# B&R Automation Studio project TD52 (part 64)

```c
    /* Switch: '<S85>/Switch' incorporates:
     *  RelationalOperator: '<S85>/UpperRelop'
     */
    if (rtb_deltafalllimit_h0 < rtb_Saturation_e) {
      rtb_Sum1_dh = rtb_Saturation_e;
    } else {
      rtb_Sum1_dh = rtb_deltafalllimit_h0;
    }

    /* End of Switch: '<S85>/Switch' */
  }

  /* End of Switch: '<S85>/Switch2' */

  /* Sum: '<S81>/Difference Inputs2' incorporates:
   *  Delay: '<S81>/Delay'
   */
  rtb_Saturation_e = rtb_Sum1_dh + Gen2_ref_DWork->Delay_DSTATE_h;

  /* Switch: '<S77>/Switch' */
  if (rtb_LogicalOperator2_p1) {
    /* Switch: '<S77>/Switch2' */
    if (Gen2_ref_B->BusInput3.traj.bRateLimRejStepSizeDep) {
      rtb_Sum1_dh = rtb_Gain_i;
    } else {
      rtb_Sum1_dh = rtb_Saturation_e;
    }

    /* End of Switch: '<S77>/Switch2' */
  } else {
    rtb_Sum1_dh = rtb_p1HP;
  }

  /* End of Switch: '<S77>/Switch' */

  /* MinMax: '<S77>/MinMax1' */
  if ((rtb_p1HP >= rtb_Sum1_dh) || rtIsNaN(rtb_Sum1_dh)) {
    rtb_MinMax1_g = rtb_p1HP;
  } else {
    rtb_MinMax1_g = rtb_Sum1_dh;
  }

  /* End of MinMax: '<S77>/MinMax1' */

  /* Abs: '<S23>/Abs1' */
  rtb_Sum1_dh = fabs(Gen2_ref_B->BusInput3.traj.rPrTriggerLargeRej);

  /* Switch: '<S23>/Switch1' incorporates:
   *  RelationalOperator: '<S23>/Relational Operator3'
   *  Sum: '<S23>/Sum7'
   */
  if (rtb_Gain_kl - rtb_p1HP > rtb_Sum1_dh) {
    rtb_Switch1_lk = Gen2_ref_B->BusInput3.traj.rTi_BDC_rej_CBV;
  } else {
    rtb_Switch1_lk = Gen2_ref_B->BusInput3.traj.rTi_BDC;
  }

  /* End of Switch: '<S23>/Switch1' */

  /* Product: '<S23>/Product1' */
  rtb_Product1_bc = Gen2_ref_B->BusInput3.traj.rFactTi_BDC_CBV * rtb_Switch1_lk;

  /* Switch: '<S1>/Switch13' incorporates:
   *  DataTypeConversion: '<S4>/Data Type Conversion16'
   */
  if (Gen2_ref_B->BusInput3.bdcMisc.bUseNsetBDC) {
    rtb_Switch13 = Gen2_ref_B->BusInput.rN_Set;
  } else {
    rtb_Switch13 = Gen2_ref_B->BusInput3.eng.rN_Nom;
  }

  /* End of Switch: '<S1>/Switch13' */

  /* Sum: '<S23>/Sum4' incorporates:
   *  Sum: '<S133>/Sum'
   */
  rtb_Switch1_kk = rtb_DataTypeConversion15 - rtb_Switch13;

  /* MATLAB Function: '<S23>/ref traj' incorporates:
   *  MATLAB Function: '<S431>/ref traj'
   *  Sum: '<S23>/Sum4'
   */
  if ((!Gen2_ref_DWork->x_not_empty_n) || rtb_LogicalOperator2_dc) {
    Gen2_ref_DWork->x_e = rtb_Gain_kl;
    Gen2_ref_DWork->x_not_empty_n = true;
    Gen2_ref_DWork->x0 = rtb_Gain_kl;
    Gen2_ref_DWork->x1 = rtb_Gain_kl;
    Gen2_ref_DWork->x2 = rtb_Gain_kl;
    Gen2_ref_DWork->x3 = rtb_Gain_kl;
    Gen2_ref_DWork->x4 = rtb_Gain_kl;
  }

  if (Gen2_ref_B->BusInput3.eng.Ts >= 0.01) {
    Ts_tmp = Gen2_ref_B->BusInput3.eng.Ts;
  } else {
    Ts_tmp = 0.01;
  }

  delta_y = rtb_MinMax1_h - rtb_Gain_kl;
  if (delta_y > Gen2_ref_B->BusInput3.traj.rThrshSwTbdcUp) {
    rtb_Switch2_j0 = Gen2_ref_B->BusInput3.traj.rTi_BDC_up;
  } else {
    rtb_Switch2_j0 = Gen2_ref_B->BusInput3.traj.rTi_BDC;
  }

  if (Gen2_ref_B->BusInput3.traj.bLimitFFcmdTV) {
    if ((rtb_Sum11 >= rtb_MinMax1_h) || rtIsNaN(rtb_MinMax1_h)) {
      FILT_IN = rtb_Sum11;
    } else {
      FILT_IN = rtb_MinMax1_h;
    }
  } else {
    FILT_IN = rtb_Sum11;
  }

  rtb_LogicalOperator5_g_tmp = rtIsNaN(Ts_tmp);
  if ((rtb_Switch2_j0 >= Ts_tmp) || rtb_LogicalOperator5_g_tmp) {
    r = rtb_Switch2_j0;
  } else {
    r = Ts_tmp;
  }

  rtb_Switch2_a = FILT_IN - Gen2_ref_DWork->x0;
  u0 = 1.0 / r * rtb_Switch2_a;
  if ((Gen2_ref_B->BusInput3.traj.rTi_BDC >= Ts_tmp) ||
      rtb_LogicalOperator5_g_tmp) {
    FILT_IN = Gen2_ref_B->BusInput3.traj.rTi_BDC;
  } else {
    FILT_IN = Ts_tmp;
  }

  u1 = 1.0 / FILT_IN * rtb_Switch2_a;
  if ((u0 >= u1) || rtIsNaN(u1)) {
    u1 = u0;
  }

  rtb_Sum10 = u1 * Ts_tmp + Gen2_ref_DWork->x0;
  if (Gen2_ref_B->BusInput3.traj.bLimitFFcmdCBV) {
    if ((rtb_Sum7_l5 >= rtb_MinMax1_g) || rtIsNaN(rtb_MinMax1_g)) {
      FILT_IN = rtb_Sum7_l5;
    } else {
      FILT_IN = rtb_MinMax1_g;
    }
  } else {
    FILT_IN = rtb_Sum7_l5;
  }

  if (rtb_Switch1_kk > 0.0) {
    if ((rtb_Switch2_j0 >= Ts_tmp) || rtb_LogicalOperator5_g_tmp) {
      r = rtb_Switch2_j0;
    } else {
      r = Ts_tmp;
    }

    rtb_Switch2_a = FILT_IN - Gen2_ref_DWork->x1;
    u0 = 1.0 / r * rtb_Switch2_a;
    if ((rtb_Product1_bc >= Ts_tmp) || rtb_LogicalOperator5_g_tmp) {
      FILT_IN = rtb_Product1_bc;
    } else {
      FILT_IN = Ts_tmp;
    }

    FILT_IN = 1.0 / FILT_IN * rtb_Switch2_a;
    if ((u0 >= FILT_IN) || rtIsNaN(FILT_IN)) {
      FILT_IN = u0;
    }
  } else {
    if ((rtb_Switch2_j0 >= Ts_tmp) || rtb_LogicalOperator5_g_tmp) {
      r = rtb_Switch2_j0;
    } else {
      r = Ts_tmp;
    }

    rtb_Switch2_a = FILT_IN - Gen2_ref_DWork->x1;
    u0 = 1.0 / r * rtb_Switch2_a;
    if ((Gen2_ref_B->BusInput3.traj.rTi_BDC >= Ts_tmp) ||
        rtb_LogicalOperator5_g_tmp) {
      FILT_IN = Gen2_ref_B->BusInput3.traj.rTi_BDC;
    } else {
      FILT_IN = Ts_tmp;
    }

    FILT_IN = 1.0 / FILT_IN * rtb_Switch2_a;
    if ((u0 >= FILT_IN) || rtIsNaN(FILT_IN)) {
      FILT_IN = u0;
    }
  }

  rtb_Switch2_h1 = FILT_IN * Ts_tmp + Gen2_ref_DWork->x1;
  if ((rtb_Switch2_j0 >= Ts_tmp) || rtb_LogicalOperator5_g_tmp) {
    r = rtb_Switch2_j0;
  } else {
    r = Ts_tmp;
  }

  rtb_Switch2_a = rtb_MinMax1_h - Gen2_ref_DWork->x2;
  u0 = 1.0 / r * rtb_Switch2_a;
  if ((Gen2_ref_B->BusInput3.traj.rTi_BDC >= Ts_tmp) ||
      rtb_LogicalOperator5_g_tmp) {
    FILT_IN = Gen2_ref_B->BusInput3.traj.rTi_BDC;
  } else {
    FILT_IN = Ts_tmp;
  }

  u1 = 1.0 / FILT_IN * rtb_Switch2_a;
  if ((u0 >= u1) || rtIsNaN(u1)) {
    u1 = u0;
  }

  rtb_Switch2_lu = u1 * Ts_tmp + Gen2_ref_DWork->x2;
  if ((rtb_Switch2_j0 >= Ts_tmp) || rtb_LogicalOperator5_g_tmp) {
    r = rtb_Switch2_j0;
  } else {
    r = Ts_tmp;
  }

  rtb_Switch2_a = rtb_MinMax1_g - Gen2_ref_DWork->x3;
  u0 = 1.0 / r * rtb_Switch2_a;
  rtb_bCBV_min = !rtb_LogicalOperator5_g_tmp;
  if ((!(rtb_Product1_bc >= Ts_tmp)) && rtb_bCBV_min) {
    rtb_Product1_bc = Ts_tmp;
  }

  u1 = 1.0 / rtb_Product1_bc * rtb_Switch2_a;
  if ((u0 >= u1) || rtIsNaN(u1)) {
    u1 = u0;
  }

  rtb_Divide3_k = u1 * Ts_tmp + Gen2_ref_DWork->x3;
  if ((rtb_Switch2_j0 >= Ts_tmp) || rtb_LogicalOperator5_g_tmp) {
    r = rtb_Switch2_j0;
  } else {
    r = Ts_tmp;
  }

  rtb_Switch2_a = rtb_Sum11 - Gen2_ref_DWork->x_e;
  u0 = 1.0 / r * rtb_Switch2_a;
  if ((Gen2_ref_B->BusInput3.traj.rTi_BDC >= Ts_tmp) ||
      rtb_LogicalOperator5_g_tmp) {
    FILT_IN = Gen2_ref_B->BusInput3.traj.rTi_BDC;
  } else {
    FILT_IN = Ts_tmp;
  }

  FILT_IN = 1.0 / FILT_IN * rtb_Switch2_a;
  if ((u0 >= FILT_IN) || rtIsNaN(FILT_IN)) {
    FILT_IN = u0;
  }

  if (FILT_IN > 0.0) {
    u0 = FILT_IN * Ts_tmp + Gen2_ref_DWork->x_e;
    rtb_Product1_bc = rtb_Gain_kl + Gen2_ref_B->BusInput3.traj.rPrR_delta_p2s;
    if ((u0 <= rtb_Product1_bc) || rtIsNaN(rtb_Product1_bc)) {
      rtb_Product1_bc = u0;
    }
  } else {
    u0 = FILT_IN * Ts_tmp + Gen2_ref_DWork->x_e;
    rtb_Product1_bc = rtb_Gain_kl - Gen2_ref_B->BusInput3.traj.rPrR_delta_p2s;
    if ((u0 >= rtb_Product1_bc) || rtIsNaN(rtb_Product1_bc)) {
      rtb_Product1_bc = u0;
    }
  }

  if ((!(rtb_Switch2_j0 >= Ts_tmp)) && rtb_bCBV_min) {
    rtb_Switch2_j0 = Ts_tmp;
  }

  rtb_Switch2_a = rtb_Sum7_l5 - Gen2_ref_DWork->x4;
  u0 = 1.0 / rtb_Switch2_j0 * rtb_Switch2_a;
  if ((!(rtb_Switch1_lk >= Ts_tmp)) && rtb_bCBV_min) {
    rtb_Switch1_lk = Ts_tmp;
  }

  u1 = 1.0 / rtb_Switch1_lk * rtb_Switch2_a;
  if (FILT_IN > 0.0) {
    if ((u0 >= u1) || rtIsNaN(u1)) {
      u1 = u0;
    }

    u0 = u1 * Ts_tmp + Gen2_ref_DWork->x4;
    rtb_Switch2_j0 = rtb_Gain_kl + Gen2_ref_B->BusInput3.traj.rPrR_delta_p2s;
    if ((u0 <= rtb_Switch2_j0) || rtIsNaN(rtb_Switch2_j0)) {
      rtb_Switch2_j0 = u0;
    }
  } else {
    if ((u0 >= u1) || rtIsNaN(u1)) {
      u1 = u0;
    }

    rtb_Switch2_j0 = u1 * Ts_tmp + Gen2_ref_DWork->x4;
  }

  Gen2_ref_DWork->x_e = rtb_Product1_bc;
  Gen2_ref_DWork->x0 = rtb_Sum10;
  Gen2_ref_DWork->x1 = rtb_Switch2_h1;
  Gen2_ref_DWork->x2 = rtb_Switch2_lu;
  Gen2_ref_DWork->x3 = rtb_Divide3_k;
  Gen2_ref_DWork->x4 = rtb_Switch2_j0;

  /* Product: '<S64>/delta rise limit' incorporates:
   *  Constant: '<S23>/Constant4'
   *  SampleTimeMath: '<S64>/sample time'
   *
   * About '<S64>/sample time':
   *  y = K where K = ( w * Ts )
   */
  rtb_Sum1_dh = 100000.0;

  /* S-Function (sfix_look1_dyn): '<S23>/Lookup Table Dynamic1' */
  /* Dynamic Look-Up Table Block: '<S23>/Lookup Table Dynamic1'
   * Input0  Data Type:  Floating Point real_T
   * Input1  Data Type:  Floating Point real_T
   * Input2  Data Type:  Floating Point real_T
   * Output0 Data Type:  Floating Point real_T
   * Lookup Method: Linear_Endpoint
   *
   */
  LookUp_real_T_real_T( &(rtb_MinMax_a),
                       &Gen2_ref_B->BusInput3.traj.rRateLimTVdpctrl[0],
                       rtb_Gain_kl, &rtb_Gain1_eu[0], 4U, inst);

  /* Abs: '<S23>/Abs3' */
  rtb_Switch1_lk = fabs(rtb_MinMax_a);

  /* Product: '<S63>/delta rise limit' incorporates:
   *  SampleTimeMath: '<S63>/sample time'
   *
   * About '<S63>/sample time':
   *  y = K where K = ( w * Ts )
   */
  rtb_MinMax_a = rtb_Switch1_lk * 0.01;

  /* Switch: '<S23>/Switch2' incorporates:
   *  Delay: '<S23>/Delay'
   *  Switch: '<S23>/Switch4'
   */
  if (Gen2_ref_DWork->Delay_DSTATE_lv) {
    FILT_IN = rtb_Product2;
  } else if (Gen2_ref_B->BusInput3.traj.bFactInitResetTVdp) {
    /* Sum: '<S23>/Sum' incorporates:
     *  MATLAB Function: '<S23>/ref traj'
     *  Switch: '<S23>/Switch4'
     */
    FILT_IN = Gen2_ref_B->BusInput3.traj.rPrR_TC_LP_min - rtb_Divide3_k;

    /* Saturate: '<S23>/Saturation' incorporates:
     *  Switch: '<S23>/Switch4'
     */
    if (FILT_IN > 1.0) {
      FILT_IN = 1.0;
    } else if (FILT_IN < 0.0) {
      FILT_IN = 0.0;
    }

    /* End of Saturate: '<S23>/Saturation' */
  } else {
    /* Switch: '<S23>/Switch4' incorporates:
     *  Constant: '<S23>/Constant2'
     */
    FILT_IN = 0.0;
  }

  /* End of Switch: '<S23>/Switch2' */

  /* Logic: '<S23>/Logical Operator4' incorporates:
   *  Constant: '<S23>/Constant1'
   *  MATLAB Function: '<S23>/ref traj'
   *  RelationalOperator: '<S23>/Relational Operator2'
   *  Sum: '<S23>/Sum4'
   */
  rtb_LogicalOperator2_p1 = (((rtb_Sum11 - rtb_Gain_kl >
    Gen2_ref_B->BusInput3.traj.rPr_delta_p2s_resetTVdp) || (delta_y >
    Gen2_ref_B->BusInput3.traj.rPr_delta_p2s_resetTVdp) ||
    rtb_LogicalOperator2_dc) && (rtb_Switch1_kk <= 0.0));

  /* Abs: '<S23>/Abs' incorporates:
   *  Sum: '<S23>/Sum4'
   */
  rtb_Switch2_a = fabs(rtb_Switch1_kk);

  /* Outputs for Atomic SubSystem: '<S23>/TON_1' */
  /* Logic: '<S23>/Logical Operator5' incorporates:
   *  Logic: '<S23>/Logical Operator6'
   *  RelationalOperator: '<S23>/Relational Operator'
   */
  Gen2_ref_TON_1(((!rtb_LogicalOperator2_p1) && (rtb_Switch2_a <=
    Gen2_ref_B->BusInput3.traj.rN_ssTVdpCtrl)),
                 Gen2_ref_B->BusInput3.traj.rT_TON_TVdpCtrl, &Gen2_ref_B->TON_1,
                 &Gen2_ref_DWork->TON_1, inst);

  /* End of Outputs for SubSystem: '<S23>/TON_1' */

  /* Switch: '<S53>/Switch' incorporates:
   *  Switch: '<S53>/Switch1'
   *  UnitDelay: '<S53>/Unit Delay4'
   */
  if (!rtb_LogicalOperator2_p1) {
    rtb_LogicalOperator2_p1 = ((!Gen2_ref_B->TON_1.LogicalOperator3) &&
      Gen2_ref_DWork->UnitDelay4_DSTATE_o);
  }

  /* End of Switch: '<S53>/Switch' */

  /* Logic: '<S23>/Logical Operator1' */
  rtb_LogicalOperator1_a0 = (rtb_LogicalOperator || rtb_LogicalOperator2_p1);

  /* Delay: '<S63>/Delay' */
  Gen2_ref_DWork->icLoad_g = ((((Gen2_ref_PrevZCSigState->Delay_Reset_ZCE_k2 ==
    1) != (int32_T)rtb_LogicalOperator1_a0) &&
    (Gen2_ref_PrevZCSigState->Delay_Reset_ZCE_k2 != 3)) ||
    rtb_LogicalOperator1_a0 || Gen2_ref_DWork->icLoad_g);
  Gen2_ref_PrevZCSigState->Delay_Reset_ZCE_k2 = rtb_LogicalOperator1_a0;
  if (Gen2_ref_DWork->icLoad_g) {
    Gen2_ref_DWork->Delay_DSTATE_c = FILT_IN;
  }

  /* Switch: '<S63>/etaVolConst' */
  if (!rtb_LogicalOperator1_a0) {
    FILT_IN = rtb_Product2;
  }

  /* End of Switch: '<S63>/etaVolConst' */

  /* Sum: '<S63>/Difference Inputs1' incorporates:
   *  Delay: '<S63>/Delay'
   */
  rtb_deltafalllimit_h0 = FILT_IN - Gen2_ref_DWork->Delay_DSTATE_c;

  /* Switch: '<S102>/Switch2' incorporates:
   *  RelationalOperator: '<S102>/LowerRelop1'
   */
  if (!(rtb_deltafalllimit_h0 > rtb_MinMax_a)) {
    /* Product: '<S63>/delta fall limit' incorporates:
     *  Gain: '<S23>/Gain4'
     *  SampleTimeMath: '<S63>/sample time'
     *
     * About '<S63>/sample time':
     *  y = K where K = ( w * Ts )
     */
    rtb_Switch1_lk = -rtb_Switch1_lk * 0.01;

    /* Switch: '<S102>/Switch' incorporates:
     *  RelationalOperator: '<S102>/UpperRelop'
     */
    if (rtb_deltafalllimit_h0 < rtb_Switch1_lk) {
      rtb_MinMax_a = rtb_Switch1_lk;
    } else {
      rtb_MinMax_a = rtb_deltafalllimit_h0;
    }

    /* End of Switch: '<S102>/Switch' */
  }

  /* End of Switch: '<S102>/Switch2' */

  /* Sum: '<S63>/Difference Inputs2' incorporates:
   *  Delay: '<S63>/Delay'
   */
  rtb_deltafalllimit_h0 = rtb_MinMax_a + Gen2_ref_DWork->Delay_DSTATE_c;

  /* Switch: '<S23>/Switch3' */
  if (rtb_LogicalOperator) {
    rtb_MinMax_a = rtb_Product2;
  } else {
    rtb_MinMax_a = rtb_deltafalllimit_h0;
  }

  /* End of Switch: '<S23>/Switch3' */

  /* Saturate: '<S23>/Saturation2' */
  if (rtb_MinMax_a <= 0.0) {
    rtb_Switch2_a = 0.0;
  } else {
    rtb_Switch2_a = rtb_MinMax_a;
  }

  /* End of Saturate: '<S23>/Saturation2' */

  /* Delay: '<S64>/Delay' incorporates:
   *  Constant: '<S23>/Constant3'
   */
  Gen2_ref_DWork->icLoad_c1 = ((((Gen2_ref_PrevZCSigState->Delay_Reset_ZCE_a ==
    1) != (int32_T)rtb_LogicalOperator2_dc) &&
    (Gen2_ref_PrevZCSigState->Delay_Reset_ZCE_a != 3)) ||
    rtb_LogicalOperator2_dc || Gen2_ref_DWork->icLoad_c1);
  Gen2_ref_PrevZCSigState->Delay_Reset_ZCE_a = rtb_LogicalOperator2_dc;
  if (Gen2_ref_DWork->icLoad_c1) {
    Gen2_ref_DWork->Delay_DSTATE_i = 0.0;
  }

  /* Switch: '<S64>/etaVolConst' incorporates:
   *  Constant: '<S23>/Constant3'
   */
  if (rtb_LogicalOperator2_dc) {
    FILT_IN = 0.0;
  } else {
    FILT_IN = rtb_Switch2_a;
  }

  /* End of Switch: '<S64>/etaVolConst' */

  /* Sum: '<S64>/Difference Inputs1' incorporates:
   *  Delay: '<S64>/Delay'
   */
  rtb_Switch1_lk = FILT_IN - Gen2_ref_DWork->Delay_DSTATE_i;

  /* Switch: '<S103>/Switch2' incorporates:
   *  RelationalOperator: '<S103>/LowerRelop1'
   */
  if (!(rtb_Switch1_lk > 100000.0)) {
    /* Product: '<S64>/delta fall limit' incorporates:
     *  Abs: '<S23>/Abs2'
     *  Gain: '<S23>/Gain7'
     *  SampleTimeMath: '<S64>/sample time'
     *
     * About '<S64>/sample time':
     *  y = K where K = ( w * Ts )
     */
    FILT_IN = -fabs(Gen2_ref_B->BusInput3.traj.rRateResetTVdpctrl) * 0.01;

    /* Switch: '<S103>/Switch' incorporates:
     *  RelationalOperator: '<S103>/UpperRelop'
     */
    if (rtb_Switch1_lk < FILT_IN) {
      rtb_Sum1_dh = FILT_IN;
    } else {
      rtb_Sum1_dh = rtb_Switch1_lk;
    }

    /* End of Switch: '<S103>/Switch' */
  }

  /* End of Switch: '<S103>/Switch2' */

  /* Sum: '<S64>/Difference Inputs2' incorporates:
   *  Delay: '<S64>/Delay'
   */
  rtb_Switch1_lk = rtb_Sum1_dh + Gen2_ref_DWork->Delay_DSTATE_i;

  /* Sum: '<S23>/Sum5' incorporates:
   *  MATLAB Function: '<S23>/ref traj'
   */
  FILT_IN = rtb_Switch2_h1 + rtb_Switch1_lk;

  /* Switch: '<S54>/Switch2' incorporates:
   *  RelationalOperator: '<S54>/LowerRelop1'
   *  RelationalOperator: '<S54>/UpperRelop'
   *  Switch: '<S54>/Switch'
   */
  if (FILT_IN > rtb_Switch2_oou) {
    rtb_Switch2_h1 = rtb_Switch2_oou;
  } else if (FILT_IN < Gen2_ref_B->BusInput3.traj.rPrMinRefp2ff) {
    /* Switch: '<S54>/Switch' */
    rtb_Switch2_h1 = Gen2_ref_B->BusInput3.traj.rPrMinRefp2ff;
  } else {
    rtb_Switch2_h1 = FILT_IN;
  }

  /* End of Switch: '<S54>/Switch2' */

  /* Switch: '<S60>/Switch2' incorporates:
   *  MATLAB Function: '<S23>/ref traj'
   *  RelationalOperator: '<S60>/LowerRelop1'
   *  RelationalOperator: '<S60>/UpperRelop'
   *  Switch: '<S60>/Switch'
   */
  if (rtb_Switch2_lu > Gen2_ref_B->BusInput3.traj.rPr_p2s_max) {
    rtb_Switch2_lu = Gen2_ref_B->BusInput3.traj.rPr_p2s_max;
  } else if (rtb_Switch2_lu < Gen2_ref_B->BusInput3.traj.rPr_p2s_min) {
    /* Switch: '<S60>/Switch' */
    rtb_Switch2_lu = Gen2_ref_B->BusInput3.traj.rPr_p2s_min;
  }

  /* End of Switch: '<S60>/Switch2' */

  /* Sum: '<S23>/Sum2' incorporates:
   *  MATLAB Function: '<S23>/ref traj'
   */
  FILT_IN = rtb_Divide3_k + rtb_Switch2_a;

  /* Switch: '<S59>/Switch2' incorporates:
   *  RelationalOperator: '<S59>/LowerRelop1'
   *  RelationalOperator: '<S59>/UpperRelop'
   *  Switch: '<S59>/Switch'
   */
  if (FILT_IN > Gen2_ref_B->BusInput3.traj.rPr_p2s_max) {
    rtb_Sum1_dh = Gen2_ref_B->BusInput3.traj.rPr_p2s_max;
  } else if (FILT_IN < Gen2_ref_B->BusInput3.traj.rPrMinRefp2ff) {
    /* Switch: '<S59>/Switch' */
    rtb_Sum1_dh = Gen2_ref_B->BusInput3.traj.rPrMinRefp2ff;
  } else {
    rtb_Sum1_dh = FILT_IN;
  }

  /* End of Switch: '<S59>/Switch2' */

  /* Abs: '<S68>/Abs' */
  rtb_Switch2_a = fabs(Gen2_ref_B->BusInput3.bdcMisc.rRefGainScheduleSL);

  /* Switch: '<S68>/Switch' incorporates:
   *  Constant: '<S68>/Constant2'
   *  RelationalOperator: '<S68>/Relational Operator'
   */
  if (2.2204460492503131E-16 >= rtb_Switch2_a) {
    FILT_IN = 2.2204460492503131E-16;
  } else {
    FILT_IN = Gen2_ref_B->BusInput3.bdcMisc.rRefGainScheduleSL;
  }

  /* End of Switch: '<S68>/Switch' */

  /* Abs: '<S67>/Abs' */
  rtb_Switch2_a = fabs(rtb_Switch13);

  /* Sum: '<S48>/Sum8' incorporates:
   *  Gain: '<S23>/Gain3'
   */
  rtb_Product4_d = 1.0E-5 * Gen2_ref_B->p2HP_filt.Switch - rtb_Switch2_oou;

  /* Switch: '<S67>/Switch' incorporates:
   *  Constant: '<S67>/Constant2'
   *  RelationalOperator: '<S67>/Relational Operator'
   */
  if (2.2204460492503131E-16 >= rtb_Switch2_a) {
    delta_y = 2.2204460492503131E-16;
  } else {
    delta_y = rtb_Switch13;
  }

  /* End of Switch: '<S67>/Switch' */

  /* Saturate: '<S48>/Saturation1' */
  if (rtb_Product4_d <= 0.0) {
    rtb_Product4_d = 0.0;
  }

  /* End of Saturate: '<S48>/Saturation1' */

  /* Product: '<S48>/Divide3' incorporates:
   *  DataTypeConversion: '<S48>/Data Type Conversion'
   *  Product: '<S48>/Divide2'
   *  RelationalOperator: '<S48>/Relational Operator2'
   */
  rtb_Divide3_k = (real_T)(Gen2_ref_B->BusInput3.LR.rN_LR_HardLim_norm > 1.0 /
    delta_y * rtb_DataTypeConversion15) * rtb_Product4_d;

  /* DiscreteIntegrator: '<S48>/Discrete-Time Integrator' */
  if (rtb_LogicalOperator2_dc ||
      (Gen2_ref_DWork->DiscreteTimeIntegrator_PrevRe_l != 0)) {
    Gen2_ref_DWork->DiscreteTimeIntegrator_DSTAT_ac = 0.0;
  }

  if (Gen2_ref_DWork->DiscreteTimeIntegrator_DSTAT_ac >= 1.0) {
    Gen2_ref_DWork->DiscreteTimeIntegrator_DSTAT_ac = 1.0;
  } else if (Gen2_ref_DWork->DiscreteTimeIntegrator_DSTAT_ac <= 0.0) {
    Gen2_ref_DWork->DiscreteTimeIntegrator_DSTAT_ac = 0.0;
  }

  /* Switch: '<S48>/Switch' incorporates:
   *  Constant: '<S48>/ON1'
   */
  if (Gen2_ref_B->BusInput3.SpeedCtrl.bSwitch_SurgeLine_LIMIT) {
    /* Sum: '<S48>/Sum12' incorporates:
     *  DiscreteIntegrator: '<S48>/Discrete-Time Integrator'
     *  Product: '<S48>/Product2'
     */
    rtb_Product4_d = rtb_Divide3_k *
      Gen2_ref_B->BusInput3.bdcMisc.rKpSurgeProtectSL +
      Gen2_ref_DWork->DiscreteTimeIntegrator_DSTAT_ac;

    /* Saturate: '<S48>/Saturation3' */
    if (rtb_Product4_d > 5.0) {
      rtb_Product4_d = 5.0;
    } else if (rtb_Product4_d < 0.0) {
      rtb_Product4_d = 0.0;
    }

    /* End of Saturate: '<S48>/Saturation3' */
  } else {
    rtb_Product4_d = 0.0;
  }

  /* End of Switch: '<S48>/Switch' */

  /* Product: '<S48>/Divide4' incorporates:
   *  Gain: '<S23>/Gain5'
   *  Product: '<S48>/Divide5'
   */
  rtb_Product4_d *= 1.0 / FILT_IN * (1.0E-5 * Gen2_ref_B->p2s_filt.Switch);

  /* Saturate: '<S23>/Saturation3' */
  if (rtb_MinMax_a >= 0.0) {
    rtb_Switch2_a = 0.0;
  } else {
    rtb_Switch2_a = rtb_MinMax_a;
  }

  /* End of Saturate: '<S23>/Saturation3' */

  /* Gain: '<S23>/Gain6' */
  rtb_Switch2_a = -rtb_Switch2_a;

  /* Sum: '<S23>/Sum9' incorporates:
   *  MATLAB Function: '<S23>/ref traj'
   *  Sum: '<S23>/Sum11'
   */
  rtb_Product1_bc = (rtb_Product1_bc + rtb_Switch2_a) + rtb_Product4_d;

  /* Switch: '<S56>/Switch2' incorporates:
   *  RelationalOperator: '<S56>/LowerRelop1'
   *  RelationalOperator: '<S56>/UpperRelop'
   *  Switch: '<S56>/Switch'
   */
  if (rtb_Product1_bc > Gen2_ref_B->BusInput3.traj.rPr_p2s_max) {
    /* BusCreator: '<S23>/Bus Creator1' */
    rtb_BusCreator1_ref_P2s_FB_TV = Gen2_ref_B->BusInput3.traj.rPr_p2s_max;
  } else if (rtb_Product1_bc < Gen2_ref_B->BusInput3.traj.rPr_p2s_min) {
    /* Switch: '<S56>/Switch' incorporates:
     *  BusCreator: '<S23>/Bus Creator1'
     */
    rtb_BusCreator1_ref_P2s_FB_TV = Gen2_ref_B->BusInput3.traj.rPr_p2s_min;
  } else {
    /* BusCreator: '<S23>/Bus Creator1' incorporates:
     *  Switch: '<S56>/Switch'
     */
    rtb_BusCreator1_ref_P2s_FB_TV = rtb_Product1_bc;
  }

  /* End of Switch: '<S56>/Switch2' */

  /* Sum: '<S23>/Sum1' incorporates:
   *  MATLAB Function: '<S23>/ref traj'
   */
  rtb_Product1_bc = rtb_Switch2_j0 + rtb_Switch1_lk;

  /* Switch: '<S55>/Switch2' incorporates:
   *  RelationalOperator: '<S55>/LowerRelop1'
   */
  if (!(rtb_Product1_bc > rtb_Switch2_oou)) {
    /* Switch: '<S55>/Switch' incorporates:
     *  RelationalOperator: '<S55>/UpperRelop'
     */
    if (rtb_Product1_bc < Gen2_ref_B->BusInput3.traj.rPrR_TC_LP_min) {
      rtb_Switch2_oou = Gen2_ref_B->BusInput3.traj.rPrR_TC_LP_min;
    } else {
      rtb_Switch2_oou = rtb_Product1_bc;
    }

    /* End of Switch: '<S55>/Switch' */
  }

  /* End of Switch: '<S55>/Switch2' */

  /* Sum: '<S23>/Sum10' incorporates:
   *  MATLAB Function: '<S23>/ref traj'
   *  Sum: '<S23>/Sum3'
   */
  rtb_Sum10 = (rtb_Sum10 + rtb_Switch2_a) + rtb_Product4_d;

  /* Switch: '<S57>/Switch2' incorporates:
   *  RelationalOperator: '<S57>/LowerRelop1'
   *  RelationalOperator: '<S57>/UpperRelop'
   *  Switch: '<S57>/Switch'
   */
  if (rtb_Sum10 > Gen2_ref_B->BusInput3.traj.rPr_p2s_max) {
    rtb_Switch2_jf = Gen2_ref_B->BusInput3.traj.rPr_p2s_max;
  } else if (rtb_Sum10 < Gen2_ref_B->BusInput3.traj.rPr_p2s_min) {
    /* Switch: '<S57>/Switch' */
    rtb_Switch2_jf = Gen2_ref_B->BusInput3.traj.rPr_p2s_min;
  } else {
    rtb_Switch2_jf = rtb_Sum10;
  }

  /* End of Switch: '<S57>/Switch2' */

  /* Outputs for Atomic SubSystem: '<S23>/Filter2' */
  /* UnitDelay: '<S23>/Unit Delay3' */
  Gen2_ref_Filter1(rtb_Switch2_jf, Gen2_ref_B->BusInput3.traj.rTiF_PrR_der,
                   Gen2_ref_DWork->UnitDelay3_DSTATE_gf, &Gen2_ref_B->Filter2,
                   &Gen2_ref_DWork->Filter2, inst);

  /* End of Outputs for SubSystem: '<S23>/Filter2' */

  /* Outputs for Atomic SubSystem: '<S23>/Filter1' */
  Gen2_ref_Filter1(rtb_Switch2_h1, Gen2_ref_B->BusInput3.traj.rTiF_PrR_der,
                   Gen2_ref_DWork->UnitDelay3_DSTATE_gf, &Gen2_ref_B->Filter1,
                   &Gen2_ref_DWork->Filter1, inst);

  /* End of Outputs for SubSystem: '<S23>/Filter1' */

  /* Outputs for Atomic SubSystem: '<S23>/Filter4' */
  Gen2_ref_Filter1(rtb_Switch2_lu, Gen2_ref_B->BusInput3.traj.rTiF_PrR_der,
                   Gen2_ref_DWork->UnitDelay3_DSTATE_gf, &Gen2_ref_B->Filter4,
                   &Gen2_ref_DWork->Filter4, inst);

  /* End of Outputs for SubSystem: '<S23>/Filter4' */

  /* BusCreator: '<S23>/Bus Creator1' */
  rtb_BusCreator1_ref_P2_FF = rtb_Sum1_dh;
  rtb_BusCreator1_ref_P2_FB_CBV = rtb_Switch2_oou;

  /* MultiPortSwitch: '<S24>/Multiport Switch' incorporates:
   *  BusCreator: '<S23>/Bus Creator1'
   */
  if ((int32_T)Gen2_ref_B->sf_MATLABFunction_f.y == 1) {
    rtb_Sum2_a1 = rtb_Switch2_jf;
  } else {
    rtb_Sum2_a1 = rtb_Switch2_lu;
  }

  /* End of MultiPortSwitch: '<S24>/Multiport Switch' */

  /* MATLAB Function: '<S44>/engine massflow2' incorporates:
   *  Gain: '<S1>/Gain9'
   *  Gain: '<S44>/rpm2rad1'
   */
  Gen2_ref_enginemassflow2(100000.0 * rtb_Sum2_a1, Gen2_ref_B->T2s_filt.Switch,
    0.10471975511965977 * rtb_Switch13, rtb_etaVolConst_lt,
    Gen2_ref_B->BusInput3.eng.rVol_Hub_Eng, &Gen2_ref_B->sf_enginemassflow2, inst);

  /* MultiPortSwitch: '<S24>/Multiport Switch1' incorporates:
   *  BusCreator: '<S23>/Bus Creator1'
   */
  if ((int32_T)Gen2_ref_B->sf_MATLABFunction_f.y == 1) {
    rtb_Sum2_a1 = Gen2_ref_B->Filter2.Switch1;
  } else {
    rtb_Sum2_a1 = Gen2_ref_B->Filter4.Switch1;
  }

  /* End of MultiPortSwitch: '<S24>/Multiport Switch1' */

  /* Gain: '<S1>/Gain10' */
  rtb_Switch2_oou = 100000.0 * rtb_Sum2_a1;

  /* DataTypeConversion: '<S155>/Data Type Conversion' */
  rtb_Sum2_a1 = Gen2_ref_B->BusInput3.bdcTv.bDynFFtv_ON;

  /* Product: '<S155>/Divide7' incorporates:
   *  Constant: '<S155>/R_air'
   */
  rtb_Product4_d = 287.15 * Gen2_ref_B->T2s_filt.Switch;

  /* Product: '<S155>/Divide6' */
  rtb_Product4_d = Gen2_ref_B->BusInput3.eng.rVol_im / rtb_Product4_d;

  /* Product: '<S155>/Divide8' */
  rtb_Switch2_oou = rtb_Switch2_oou * rtb_Sum2_a1 * rtb_Product4_d;

  /* Saturate: '<S44>/Saturation1' */
  if (Gen2_ref_B->BusInput3.eng.rNum_TV > 10.0) {
    rtb_Sum2_a1 = 10.0;
  } else if (Gen2_ref_B->BusInput3.eng.rNum_TV < 1.0) {
    rtb_Sum2_a1 = 1.0;
  } else {
    rtb_Sum2_a1 = Gen2_ref_B->BusInput3.eng.rNum_TV;
  }

  /* End of Saturate: '<S44>/Saturation1' */

  /* Product: '<S44>/Divide' incorporates:
   *  Sum: '<S44>/Sum3'
   */
  rtb_Divide_n0 = (Gen2_ref_B->sf_enginemassflow2.dm_e + rtb_Switch2_oou) /
    rtb_Sum2_a1;

  /* MultiPortSwitch: '<S24>/Multiport Switch2' incorporates:
   *  BusCreator: '<S23>/Bus Creator1'
   */
  rtb_Sum2_a1 = rtb_Sum1_dh;

  /* Gain: '<S1>/Gain11' */
  rtb_Switch2_oou = 100000.0 * rtb_Sum2_a1;

  /* MultiPortSwitch: '<S24>/Multiport Switch3' incorporates:
   *  BusCreator: '<S23>/Bus Creator1'
   */
  rtb_Sum2_a1 = rtb_Switch2_lu;

  /* Gain: '<S1>/Gain12' */
  rtb_Sum10 = 100000.0 * rtb_Sum2_a1;

  /* MATLAB Function: '<S44>/MATLAB Function3' incorporates:
   *  Constant: '<S44>/Constant3'
   *  Product: '<S44>/Product1'
   */
  if (rtb_Switch2_oou >= rtb_Sum10) {
    r = rtb_Sum10 / rtb_Switch2_oou;
    if ((1.0E-6 >= r) || rtIsNaN(r)) {
      r = 1.0E-6;
    }

    if (1.0 / r <= 1.8929291587378541) {
      u0 = 0.78539816339744828 * Gen2_ref_B->BusInput3.bdcTv.rDref *
        Gen2_ref_B->BusInput3.bdcTv.rDref * rtb_Switch2_oou / sqrt(287.15 *
        Gen2_ref_B->T2s_filt.Switch) * sqrt((rt_powd_snf(r, 1.4285714285714286, inst)
        - rt_powd_snf(r, 1.7142857142857144, inst)) * 7.0000000000000009);
      if (!(u0 >= 1.0E-6)) {
        u0 = 1.0E-6;
      }

      rtb_Switch2_oou = rtb_Divide_n0 / u0;
    } else {
      u0 = 0.78539816339744828 * Gen2_ref_B->BusInput3.bdcTv.rDref *
        Gen2_ref_B->BusInput3.bdcTv.rDref * rtb_Switch2_oou / sqrt(287.15 *
        Gen2_ref_B->T2s_filt.Switch) * 0.6847314563772704;
      if (!(u0 >= 1.0E-6)) {
        u0 = 1.0E-6;
      }

      rtb_Switch2_oou = rtb_Divide_n0 / u0;
    }
  } else {
    rtb_Switch2_oou = 1.0;
  }

  /* End of MATLAB Function: '<S44>/MATLAB Function3' */

  /* Saturate: '<S44>/Saturation3' */
  if (rtb_Switch2_oou > 1.0) {
    rtb_Sum2_a1 = 1.0;
  } else if (rtb_Switch2_oou < 0.0) {
    rtb_Sum2_a1 = 0.0;
  } else {
    rtb_Sum2_a1 = rtb_Switch2_oou;
  }

  /* End of Saturate: '<S44>/Saturation3' */

  /* S-Function (sfix_look1_dyn): '<S44>/Lookup Table Dynamic1' */
  /* Dynamic Look-Up Table Block: '<S44>/Lookup Table Dynamic1'
   * Input0  Data Type:  Floating Point real_T
   * Input1  Data Type:  Floating Point real_T
   * Input2  Data Type:  Floating Point real_T
   * Output0 Data Type:  Floating Point real_T
   * Lookup Method: Linear_Endpoint
   *
   */
  LookUp_real_T_real_T( &(rtb_Product4_d),
                       &Gen2_ref_B->BusInput3.bdcTv.rCd_vect_x[0], rtb_Sum2_a1,
                       &Gen2_ref_B->BusInput3.bdcTv.rCd_vect_y[0], 10U, inst);

  /* MinMax: '<S44>/MinMax' */
  rtb_Sum1_dh = Gen2_ref_B->BusInput3.bdcTv.rCd_vect_x[0];
  for (k = 0; k < 10; k++) {
    u1 = Gen2_ref_B->BusInput3.bdcTv.rCd_vect_x[k + 1];
    if ((!(rtb_Sum1_dh >= u1)) && (!rtIsNaN(u1))) {
      rtb_Sum1_dh = u1;
    }
  }

  /* End of MinMax: '<S44>/MinMax' */

  /* Switch: '<S154>/Switch' incorporates:
   *  Abs: '<S154>/Abs'
   *  Constant: '<S154>/Constant2'
   *  RelationalOperator: '<S154>/Relational Operator'
   */
  if (2.2204460492503131E-16 >= fabs(rtb_Sum1_dh)) {
    rtb_Sum1_dh = 2.2204460492503131E-16;
  }

  /* End of Switch: '<S154>/Switch' */

  /* Product: '<S44>/Divide1' */
  rtb_Switch2_oou = rtb_Product4_d / rtb_Sum1_dh;

  /* Saturate: '<S44>/Saturation' */
  rtb_Product4_d = rtb_Saturation1_i;

  /* Product: '<S44>/Product' */
  rtb_Switch2_oou *= rtb_Product4_d;

  /* Gain: '<S427>/Gain1' */
  rtb_Product4_d = 0.001 * Gen2_ref_B->BusInput3.LR.rTi_LR_LIM_TV_OFF;

  /* Outputs for Atomic SubSystem: '<S427>/TOF3' */
  /* Logic: '<S427>/Logical Operator14' incorporates:
   *  Bias: '<S427>/ u+Ts3'
   *  Logic: '<S427>/Logical Operator15'
   *  RelationalOperator: '<S427>/Relational Operator10'
   *  RelationalOperator: '<S427>/Relational Operator5'
   */
  Gen2_ref_TOF((rtb_RelationalOperator2_j &&
                Gen2_ref_B->BusInput3.LR.bLIM_TVbyP2s_OFFatLargeRej &&
                ((rtb_Saturation > Gen2_ref_B->BusInput3.LR.rP_Trig_TVbyP2S_OFF)
                 || (rtb_Divide4_d > Gen2_ref_B->BusInput3.LR.rN_LR_HardLim_norm))),
               rtb_Product4_d + 0.01, &Gen2_ref_B->TOF3, &Gen2_ref_DWork->TOF3, inst);

  /* End of Outputs for SubSystem: '<S427>/TOF3' */

  /* Logic: '<S427>/Logical Operator16' incorporates:
   *  Logic: '<S427>/Logical Operator17'
   *  RelationalOperator: '<S427>/Relational Operator7'
   *  UnitDelay: '<S427>/Unit Delay1'
   */
  rtb_LogicalOperator1_a0 = (Gen2_ref_B->TOF3.LogicalOperator1 ||
    ((rtb_Divide4_d > Gen2_ref_B->BusInput3.LR.rN_LIM_TVbyPOS_ON) &&
     Gen2_ref_DWork->UnitDelay1_DSTATE_m));

  /* Switch: '<S133>/Switch' incorporates:
   *  Logic: '<S43>/Logical Operator'
   *  Switch: '<S133>/Switch1'
   */
  if (rtb_LogicalOperator1_a0) {
    rtb_Switch_e = Gen2_ref_B->BusInput3.bdcTv.rPos_min;
  } else {
    if (Gen2_ref_B->BusInput3.LR.bSwitch_Surge_TV_Min) {
      /* Gain: '<S133>/Gain1' incorporates:
       *  Switch: '<S133>/Switch1'
       */
      rtb_Sum10 = rtb_kW2W1_h;

      /* S-Function (sfix_look1_dyn): '<S133>/Surge protection depending  on boost pressure' incorporates:
       *  Switch: '<S133>/Switch1'
       */
      /* Dynamic Look-Up Table Block: '<S133>/Surge protection depending  on boost pressure'
       * Input0  Data Type:  Floating Point real_T
       * Input1  Data Type:  Floating Point real_T
       * Input2  Data Type:  Floating Point real_T
       * Output0 Data Type:  Floating Point real_T
       * Lookup Method: Linear_Endpoint
       *
       */
      LookUp_real_T_real_T( &(rtb_Surgeprotectiondependingonb),
                           &Gen2_ref_B->BusInput3.LR.rLCRCurve_DK_min_Lup_y[0],
                           rtb_Sum10,
                           &Gen2_ref_B->BusInput3.LR.rLCRCurve_DK_min_Lup_x[0],
                           7U, inst);

      /* Switch: '<S133>/Switch1' incorporates:
       *  Sum: '<S133>/Sum1'
       */
      rtb_Sum10 = rtb_Surgeprotectiondependingonb +
        Gen2_ref_B->BusInput3.LR.rLCRCurve_DK_min_Lup_offset;
    } else {
      /* Switch: '<S133>/Switch1' */
      rtb_Sum10 = Gen2_ref_B->BusInput3.bdcTv.rPos_min;
    }

    /* Switch: '<S136>/Switch2' incorporates:
     *  RelationalOperator: '<S136>/LowerRelop1'
     *  RelationalOperator: '<S136>/UpperRelop'
     *  Switch: '<S136>/Switch'
     */
    if (rtb_Sum10 > Gen2_ref_B->BusInput3.bdcTv.rPos_max) {
      rtb_Switch_e = Gen2_ref_B->BusInput3.bdcTv.rPos_max;
    } else if (rtb_Sum10 < Gen2_ref_B->BusInput3.bdcTv.rPos_min) {
      /* Switch: '<S136>/Switch' */
      rtb_Switch_e = Gen2_ref_B->BusInput3.bdcTv.rPos_min;
    } else {
      rtb_Switch_e = rtb_Sum10;
    }

    /* End of Switch: '<S136>/Switch2' */
  }

  /* Switch: '<S157>/Switch2' incorporates:
   *  RelationalOperator: '<S157>/LowerRelop1'
   *  RelationalOperator: '<S157>/UpperRelop'
   *  Switch: '<S157>/Switch'
   */
  if (rtb_Switch2_oou > Gen2_ref_B->BusInput3.bdcTv.rPos_max) {
    rtb_Product4_d = Gen2_ref_B->BusInput3.bdcTv.rPos_max;
  } else if (rtb_Switch2_oou < rtb_Switch_e) {
    /* Switch: '<S157>/Switch' */
    rtb_Product4_d = rtb_Switch_e;
  } else {
    rtb_Product4_d = rtb_Switch2_oou;
  }

  /* End of Switch: '<S157>/Switch2' */

  /* Switch: '<S45>/Switch4' incorporates:
   *  Constant: '<S45>/Constant1'
   */
  if (Gen2_ref_B->BusInput3.bdcTv.bActive_ff) {
    rtb_Sum1_dh = rtb_Product4_d;
  } else {
    rtb_Sum1_dh = 0.0;
  }

  /* End of Switch: '<S45>/Switch4' */

  /* Saturate: '<S45>/Saturation1' */
  if (rtb_Sum1_dh > 1.0) {
    rtb_Switch2_oou = 1.0;
  } else if (rtb_Sum1_dh < 0.0) {
    rtb_Switch2_oou = 0.0;
  } else {
    rtb_Switch2_oou = rtb_Sum1_dh;
  }

  /* End of Saturate: '<S45>/Saturation1' */

  /* Outputs for Atomic SubSystem: '<S45>/Inverse_Linearization1' */
  Gen2_ref_Inverse_Linearization4(rtb_Switch2_oou, &Gen2_ref_B->BusInput3,
    &Gen2_ref_B->Inverse_Linearization1, inst);

  /* End of Outputs for SubSystem: '<S45>/Inverse_Linearization1' */

  /* S-Function (sfix_look1_dyn): '<S41>/Lookup8' */
  /* Dynamic Look-Up Table Block: '<S41>/Lookup8'
   * Input0  Data Type:  Floating Point real_T
   * Input1  Data Type:  Floating Point real_T
   * Input2  Data Type:  Floating Point real_T
   * Output0 Data Type:  Floating Point real_T
   * Lookup Method: Linear_Endpoint
   *
   */
  LookUp_real_T_real_T( &(rtb_Sum1_dh),
                       &Gen2_ref_B->BusInput3.bdcTv.rGainMultRej_y[0],
                       rtb_DataTypeConversion15,
                       &Gen2_ref_B->BusInput3.bdcTv.rGainMultRej_x[0], 4U, inst);

  /* Gain: '<S41>/Pa2bar' incorporates:
   *  DiscreteIntegrator: '<S132>/Discrete-Time Integrator'
   */
  rtb_Pa2bar = 1.0E-5 * Gen2_ref_DWork->DiscreteTimeIntegrator_DSTATE_g;

  /* Switch: '<S41>/Switch11' incorporates:
   *  Sum: '<S41>/Sum2'
   *  Sum: '<S41>/Sum4'
   */
  if (rtb_LogicalOperator) {
    /* S-Function (sfix_look1_dyn): '<S41>/Lookup' */
    /* Dynamic Look-Up Table Block: '<S41>/Lookup'
     * Input0  Data Type:  Floating Point real_T
     * Input1  Data Type:  Floating Point real_T
     * Input2  Data Type:  Floating Point real_T
     * Output0 Data Type:  Floating Point real_T
     * Lookup Method: Linear_Endpoint
     *
     */
    LookUp_real_T_real_T( &(rtb_kp_m), &Gen2_ref_B->BusInput3.bdcTv.rKp_Lup[0],
                         rtb_Pa2bar, &Gen2_ref_B->BusInput3.bdcMisc.rPr_Lup_in[0],
                         9U, inst);
    rtb_Switch2_oou = rtb_kp_m + Gen2_ref_B->BusInput3.bdcTv.rKp_grid_offset;
  } else {
    /* S-Function (sfix_look1_dyn): '<S41>/Lookup1' */
    /* Dynamic Look-Up Table Block: '<S41>/Lookup1'
     * Input0  Data Type:  Floating Point real_T
     * Input1  Data Type:  Floating Point real_T
     * Input2  Data Type:  Floating Point real_T
     * Output0 Data Type:  Floating Point real_T
     * Lookup Method: Linear_Endpoint
     *
     */
    LookUp_real_T_real_T( &(rtb_Lookup1),
                         &Gen2_ref_B->BusInput3.bdcTv.rKp_island_Lup[0],
                         rtb_Pa2bar, &Gen2_ref_B->BusInput3.bdcMisc.rPr_Lup_in[0],
                         9U, inst);
    rtb_Switch2_oou = rtb_Lookup1 +
      Gen2_ref_B->BusInput3.bdcTv.rKp_island_offset;
  }

  /* End of Switch: '<S41>/Switch11' */

  /* Product: '<S41>/Product' */
  rtb_Switch2_oou *= rtb_Sum1_dh;

  /* Switch: '<S128>/Switch2' incorporates:
   *  RelationalOperator: '<S128>/LowerRelop1'
   *  RelationalOperator: '<S128>/UpperRelop'
   *  Switch: '<S128>/Switch'
   */
  if (rtb_Switch2_oou > Gen2_ref_B->BusInput3.bdcMisc.rKpMax) {
    FILT_IN = Gen2_ref_B->BusInput3.bdcMisc.rKpMax;
  } else if (rtb_Switch2_oou < Gen2_ref_B->BusInput3.bdcMisc.rKpMin) {
    /* Switch: '<S128>/Switch' */
    FILT_IN = Gen2_ref_B->BusInput3.bdcMisc.rKpMin;
  } else {
    FILT_IN = rtb_Switch2_oou;
  }

  /* End of Switch: '<S128>/Switch2' */

  /* DataTypeConversion: '<S1>/Data Type Conversion20' */
  rtb_Sum1_dh = Gen2_ref_B->BusInput3.bdcMisc.bActive_BDC;

  /* Logic: '<S1>/Logical Operator' incorporates:
   *  DataTypeConversion: '<S1>/Data Type Conversion12'
   */
  rtb_LogicalOperator3_k = !(rtb_Sum1_dh != 0.0);

  /* MATLAB Function: '<S45>/tv_fb_err' incorporates:
   *  BusCreator: '<S23>/Bus Creator1'
   *  SignalConversion generated from: '<S168>/ SFunction '
   */
  if ((!Gen2_ref_DWork->err_1_not_empty) || rtb_LogicalOperator3_k) {
    Gen2_ref_DWork->err_1 = 0.0;
    Gen2_ref_DWork->err_1_not_empty = true;
  }

  rtb_Sum10 = rtb_BusCreator1_ref_P2s_FB_TV - rtb_Divide3_a0;
  rtb_i_reset = (Gen2_ref_B->BusInput.tLvrt.bLvrtFlg || rtb_LogicalOperator3_k);
  rtb_Switch2_oou = Gen2_ref_DWork->err_1 - rtb_Sum10;
  Gen2_ref_DWork->err_1 = rtb_Sum10;

  /* Product: '<S45>/Product4' incorporates:
   *  MATLAB Function: '<S45>/tv_fb_err'
   */
  rtb_Product4 = FILT_IN * rtb_Sum10;

  /* Logic: '<S45>/Logical Operator1' incorporates:
   *  Logic: '<S45>/Logical Operator2'
   *  RelationalOperator: '<S160>/FixPt Relational Operator'
   *  UnitDelay: '<S160>/Delay Input1'
   */
  rtb_bCBV_min = ((Gen2_ref_B->BusInput3.bdcTv.bActive_ff !=
                   Gen2_ref_DWork->DelayInput1_DSTATE_f) &&
                  ((!rtb_LogicalOperator3_k) && rtb_LogicalOperator_b));

  /* Logic: '<S45>/Logical Operator3' */
  rtb_LogicalOperator3_aa = (rtb_i_reset || rtb_bCBV_min);

  /* Delay: '<S45>/Delay' */
  if (Gen2_ref_DWork->icLoad_eh) {
    Gen2_ref_DWork->Delay_DSTATE_cn =
      Gen2_ref_B->Inverse_Linearization1.LCRScal_Lam_EOT1;
  }

  /* Outputs for Atomic SubSystem: '<S161>/Inverse_Linearization4' */
  Gen2_ref_Inverse_Linearization4(Gen2_ref_B->BusInput3.bdcTv.rPos_Start,
    &Gen2_ref_B->BusInput3, &Gen2_ref_B->Inverse_Linearization4, inst);

  /* End of Outputs for SubSystem: '<S161>/Inverse_Linearization4' */

  /* Sum: '<S161>/Add2' */
  rtb_Add2 = (Gen2_ref_B->Inverse_Linearization4.LCRScal_Lam_EOT1 -
              Gen2_ref_B->Inverse_Linearization1.LCRScal_Lam_EOT1) -
    rtb_Product4;

  /* Delay: '<S161>/Delay' */
  if ((((Gen2_ref_PrevZCSigState->Delay_Reset_ZCE_o == 1) != (int32_T)
        rtb_LogicalOperator3_k) && (Gen2_ref_PrevZCSigState->Delay_Reset_ZCE_o
        != 3)) || rtb_LogicalOperator3_k) {
    Gen2_ref_DWork->Delay_DSTATE_gp = 0.0;
  }

  Gen2_ref_PrevZCSigState->Delay_Reset_ZCE_o = rtb_LogicalOperator3_k;

  /* Switch: '<S45>/Switch1' incorporates:
   *  Delay: '<S161>/Delay2'
   *  Delay: '<S45>/Delay'
   *  Sum: '<S45>/Sum'
   *  Sum: '<S45>/Sum4'
   *  Switch: '<S161>/Switch1'
   *  Switch: '<S161>/Switch3'
   *  UnitDelay: '<S45>/Unit Delay1'
   */
  if (rtb_bCBV_min) {
    rtb_Switch1_d2 = (Gen2_ref_DWork->Delay_DSTATE_cn -
                      Gen2_ref_B->Inverse_Linearization1.LCRScal_Lam_EOT1) +
      Gen2_ref_DWork->UnitDelay1_DSTATE_ed;
  } else if (Gen2_ref_DWork->Delay2_DSTATE_f) {
    /* Switch: '<S161>/Switch3' */
    rtb_Switch1_d2 = rtb_Add2;
  } else if (Gen2_ref_B->BusInput.tLvrt.bLvrtFlg) {
    /* Outputs for Atomic SubSystem: '<S45>/Inverse_Linearization4' */
    /* S-Function (sfix_look1_dyn): '<S165>/LCRScal_Lam_EOT1' incorporates:
     *  Switch: '<S161>/Switch1'
     *  Switch: '<S161>/Switch3'
     */
    /* Dynamic Look-Up Table Block: '<S165>/LCRScal_Lam_EOT1'
     * Input0  Data Type:  Floating Point real32_T
     * Input1  Data Type:  Floating Point real_T
     * Input2  Data Type:  Floating Point real_T
     * Output0 Data Type:  Floating Point real_T
     * Lookup Method: Linear_Endpoint
     *
     */
    LookUp_real_T_real32_Treal_T( &(rtb_LCRScal_Lam_EOT1_i),
      &Gen2_ref_B->BusInput3.bdcTv.rPosTv_Lin_x[0],
      Gen2_ref_B->BusInput.tLvrt.rTvPosFb,
      &Gen2_ref_B->BusInput3.bdcTv.rPosTv_Lin_y[0], 9U, inst);

    /* End of Outputs for SubSystem: '<S45>/Inverse_Linearization4' */

    /* Switch: '<S161>/Switch1' incorporates:
     *  Sum: '<S161>/Add3'
     *  Switch: '<S161>/Switch3'
     */
    rtb_Switch1_d2 = (rtb_LCRScal_Lam_EOT1_i -
                      Gen2_ref_B->Inverse_Linearization1.LCRScal_Lam_EOT1) -
      rtb_Product4;
  } else {
    /* Switch: '<S161>/Switch1' incorporates:
     *  Delay: '<S161>/Delay'
     *  Delay: '<S161>/Delay1'
     *  Product: '<S45>/Product3'
     *  Sum: '<S161>/Add1'
     *  Switch: '<S161>/Switch3'
     */
    rtb_Switch1_d2 = (rtb_Switch2_oou * FILT_IN +
                      Gen2_ref_DWork->Delay1_DSTATE_l) +
      Gen2_ref_DWork->Delay_DSTATE_gp;
  }

  /* End of Switch: '<S45>/Switch1' */

  /* DiscreteIntegrator: '<S45>/Discrete-Time Integrator1' */
  if (Gen2_ref_DWork->DiscreteTimeIntegrator1_IC_LOAD != 0) {
    Gen2_ref_DWork->DiscreteTimeIntegrator1_DSTAT_n = rtb_Switch1_d2;
  }

  if (rtb_LogicalOperator3_aa ||
      (Gen2_ref_DWork->DiscreteTimeIntegrator1_PrevR_k != 0)) {
    Gen2_ref_DWork->DiscreteTimeIntegrator1_DSTAT_n = rtb_Switch1_d2;
  }

  rtb_Product1_bc = Gen2_ref_DWork->DiscreteTimeIntegrator1_DSTAT_n;

  /* Sum: '<S45>/Sum2' incorporates:
   *  DiscreteIntegrator: '<S45>/Discrete-Time Integrator1'
   */
  rtb_Switch2_oou = rtb_Product4 +
    Gen2_ref_DWork->DiscreteTimeIntegrator1_DSTAT_n;

  /* BusCreator: '<Root>/Bus Creator' incorporates:
   *  BusCreator: '<S45>/Bus Creator'
   *  DataTypeConversion: '<S45>/Data Type Conversion1'
   *  Outport: '<Root>/dbg'
   */
  Gen2_ref_Y->dbg.BDC.tv.fb = (real32_T)rtb_Switch2_oou;

  /* Sum: '<S45>/Sum5' */
  rtb_Switch2_a = Gen2_ref_B->Inverse_Linearization1.LCRScal_Lam_EOT1 +
    rtb_Switch2_oou;

  /* MinMax: '<S45>/MinMax' */
  if ((Gen2_ref_B->BusInput3.bdcTv.rPos_min >= rtb_Switch_e) || rtIsNaN
      (rtb_Switch_e)) {
    delta_y = Gen2_ref_B->BusInput3.bdcTv.rPos_min;
  } else {
    delta_y = rtb_Switch_e;
  }

  /* End of MinMax: '<S45>/MinMax' */

  /* Outputs for Atomic SubSystem: '<S45>/Inverse_Linearization3' */
  Gen2_ref_Inverse_Linearization4(delta_y, &Gen2_ref_B->BusInput3,
    &Gen2_ref_B->Inverse_Linearization3, inst);

  /* End of Outputs for SubSystem: '<S45>/Inverse_Linearization3' */

  /* Outputs for Atomic SubSystem: '<S427>/TP_ActSat_TV' */
  /* Logic: '<S427>/Logical Operator2' incorporates:
   *  Bias: '<S427>/u+Ts1'
   *  Delay: '<S427>/Delay'
   *  Gain: '<S427>/Gain4'
   *  RelationalOperator: '<S427>/Relational Operator16'
   *  RelationalOperator: '<S427>/Relational Operator17'
   */
  Gen2_ref_TP_ActSat_CBV((rtb_RelationalOperator2_j &&
    Gen2_ref_B->BusInput3.LR.bP_LoadReject_Active &&
    (Gen2_ref_DWork->Delay_DSTATE[0] >=
     Gen2_ref_B->BusInput3.LR.rP_LR_Trig_ActSat_TV) && (rtb_Saturation >
    Gen2_ref_B->BusInput3.LR.rP_LR_Trig_ActSat_TV) &&
    Gen2_ref_B->BusInput3.LR.bLR_ActSat_TV), 0.001 *
    Gen2_ref_B->BusInput3.LR.rTi_LR_ActSat_TV + 0.01, &Gen2_ref_B->TP_ActSat_TV,
    &Gen2_ref_DWork->TP_ActSat_TV, inst);

  /* End of Outputs for SubSystem: '<S427>/TP_ActSat_TV' */

  /* Switch: '<S45>/Switch2' */
  if (Gen2_ref_B->TP_ActSat_TV.LogicalOperator1) {
    rtb_Switch2_by = Gen2_ref_B->Inverse_Linearization3.LCRScal_Lam_EOT1;
  } else {
    /* Outputs for Atomic SubSystem: '<S45>/Inverse_Linearization2' */
    Gen2_ref_Inverse_Linearization4(Gen2_ref_B->BusInput3.bdcTv.rPos_max,
      &Gen2_ref_B->BusInput3, &Gen2_ref_B->Inverse_Linearization2, inst);

    /* End of Outputs for SubSystem: '<S45>/Inverse_Linearization2' */

    /* Switch: '<S167>/Switch2' incorporates:
     *  RelationalOperator: '<S167>/LowerRelop1'
     *  RelationalOperator: '<S167>/UpperRelop'
     *  Switch: '<S167>/Switch'
     */
    if (rtb_Switch2_a > Gen2_ref_B->Inverse_Linearization2.LCRScal_Lam_EOT1) {
      rtb_Switch2_by = Gen2_ref_B->Inverse_Linearization2.LCRScal_Lam_EOT1;
    } else if (rtb_Switch2_a <
               Gen2_ref_B->Inverse_Linearization3.LCRScal_Lam_EOT1) {
      /* Switch: '<S167>/Switch' */
      rtb_Switch2_by = Gen2_ref_B->Inverse_Linearization3.LCRScal_Lam_EOT1;
    } else {
      rtb_Switch2_by = rtb_Switch2_a;
    }

    /* End of Switch: '<S167>/Switch2' */
  }

  /* End of Switch: '<S45>/Switch2' */

  /* Switch: '<S41>/Switch4' incorporates:
   *  Constant: '<S41>/Constant1'
   *  Gain: '<S41>/Pa2bar1'
   *  RelationalOperator: '<S41>/Relational Operator'
   *  RelationalOperator: '<S41>/Relational Operator1'
   *  Sum: '<S41>/Sum8'
   *  Sum: '<S41>/Sum9'
   *  UnitDelay: '<S41>/Unit Delay'
   */
  if (rtb_DataTypeConversion15 < 0.5 *
      Gen2_ref_B->BusInput3.SpeedCtrl.rOutOfNWindow + rtb_Switch13) {
    rtb_Switch4_j = false;
  } else {
    rtb_Switch4_j = ((rtb_DataTypeConversion15 >
                      Gen2_ref_B->BusInput3.SpeedCtrl.rOutOfNWindow +
                      rtb_Switch13) || Gen2_ref_DWork->UnitDelay_DSTATE_je);
  }

  /* End of Switch: '<S41>/Switch4' */

  /* Switch: '<S41>/Switch1' incorporates:
   *  Sum: '<S41>/Sum3'
   *  Sum: '<S41>/Sum5'
   */
  if (rtb_LogicalOperator) {
    /* S-Function (sfix_look1_dyn): '<S41>/Lookup2' */
    /* Dynamic Look-Up Table Block: '<S41>/Lookup2'
     * Input0  Data Type:  Floating Point real_T
     * Input1  Data Type:  Floating Point real_T
     * Input2  Data Type:  Floating Point real_T
     * Output0 Data Type:  Floating Point real_T
     * Lookup Method: Linear_Endpoint
     *
     */
    LookUp_real_T_real_T( &(rtb_Lookup2), &Gen2_ref_B->BusInput3.bdcTv.rKi_Lup[0],
                         rtb_Pa2bar, &Gen2_ref_B->BusInput3.bdcMisc.rPr_Lup_in[0],
                         9U, inst);
    rtb_Switch2_oou = rtb_Lookup2 + Gen2_ref_B->BusInput3.bdcTv.rKi_grid_offset;
  } else {
    /* Logic: '<S41>/Logical Operator1' */
    rtb_LogicalOperator1_ix = (rtb_Switch4_j &&
      Gen2_ref_B->BusInput3.bdcTv.bKi_island_reject);

    /* Switch: '<S41>/Switch6' */
    for (i = 0; i < 10; i++) {
      if (rtb_LogicalOperator1_ix) {
        rtb_Switch6_n[i] = Gen2_ref_B->BusInput3.bdcTv.rKi_island_reject_Lup[i];
      } else {
        rtb_Switch6_n[i] = Gen2_ref_B->BusInput3.bdcTv.rKi_island_Lup[i];
      }
    }

    /* End of Switch: '<S41>/Switch6' */

    /* S-Function (sfix_look1_dyn): '<S41>/Lookup3' */
    /* Dynamic Look-Up Table Block: '<S41>/Lookup3'
     * Input0  Data Type:  Floating Point real_T
     * Input1  Data Type:  Floating Point real_T
     * Input2  Data Type:  Floating Point real_T
     * Output0 Data Type:  Floating Point real_T
     * Lookup Method: Linear_Endpoint
     *
     */
    LookUp_real_T_real_T( &(rtb_Lookup3), &rtb_Switch6_n[0], rtb_Pa2bar,
                         &Gen2_ref_B->BusInput3.bdcMisc.rPr_Lup_in[0], 9U, inst);
    rtb_Switch2_oou = rtb_Lookup3 +
      Gen2_ref_B->BusInput3.bdcTv.rKi_island_offset;
  }

  /* End of Switch: '<S41>/Switch1' */

  /* Switch: '<S129>/Switch2' incorporates:
   *  RelationalOperator: '<S129>/LowerRelop1'
   *  RelationalOperator: '<S129>/UpperRelop'
   *  Switch: '<S129>/Switch'
   */
  if (rtb_Switch2_oou > Gen2_ref_B->BusInput3.bdcMisc.rKiMax) {
    rtb_Switch2_j0 = Gen2_ref_B->BusInput3.bdcMisc.rKiMax;
  } else if (rtb_Switch2_oou < Gen2_ref_B->BusInput3.bdcMisc.rKiMin) {
    /* Switch: '<S129>/Switch' */
    rtb_Switch2_j0 = Gen2_ref_B->BusInput3.bdcMisc.rKiMin;
  } else {
    rtb_Switch2_j0 = rtb_Switch2_oou;
  }

  /* End of Switch: '<S129>/Switch2' */

  /* Switch: '<S45>/Switch5' incorporates:
   *  Constant: '<S45>/Constant3'
   *  Product: '<S45>/Divide'
   *  RelationalOperator: '<S45>/Relational Operator'
   */
  if (Gen2_ref_B->BusInput3.bdcTv.rKaw <= 0.0) {
    /* Saturate: '<S45>/Saturation' */
    if (FILT_IN <= 0.1) {
      FILT_IN = 0.1;
    }

    /* End of Saturate: '<S45>/Saturation' */
    rtb_Switch2_oou = rtb_Switch2_j0 / FILT_IN;
  } else {
    rtb_Switch2_oou = Gen2_ref_B->BusInput3.bdcTv.rKaw;
  }

  /* End of Switch: '<S45>/Switch5' */

  /* Product: '<S45>/Product2' incorporates:
   *  Sum: '<S45>/Sum1'
   */
  rtb_Switch2_oou *= rtb_Switch2_by - rtb_Switch2_a;

  /* BusCreator: '<Root>/Bus Creator' incorporates:
   *  BusCreator: '<S45>/Bus Creator'
   *  DataTypeConversion: '<S45>/Data Type Conversion5'
   *  Outport: '<Root>/dbg'
   */
  Gen2_ref_Y->dbg.BDC.tv.ff_unsat = (real32_T)rtb_Product4_d;

  /* MATLAB Function: '<S25>/MATLAB Function' incorporates:
   *  Gain: '<S25>/Gain'
   *  Sum: '<S25>/Sum'
   */
  Gen2_ref_MATLABFunction(1.0E-5 * Gen2_ref_B->p2s_filt.Switch,
    Gen2_ref_B->BusInput3.bdcMisc.rPrSwitchFFmethod,
    Gen2_ref_B->BusInput3.bdcMisc.rPrSwitchFFmethod +
    Gen2_ref_B->BusInput3.bdcMisc.rPrSwitchFFmethod_hys,
    &Gen2_ref_B->sf_MATLABFunction_e, &Gen2_ref_DWork->sf_MATLABFunction_e, inst);

  /* MultiPortSwitch: '<S25>/Multiport Switch' incorporates:
   *  BusCreator: '<S23>/Bus Creator1'
   */
  if ((int32_T)Gen2_ref_B->sf_MATLABFunction_e.y == 1) {
    rtb_MultiportSwitch = rtb_Switch2_jf;
  } else {
    rtb_MultiportSwitch = rtb_Switch2_lu;
  }

  /* End of MultiPortSwitch: '<S25>/Multiport Switch' */

  /* Gain: '<S1>/Gain' */
  FILT_IN = 100000.0 * rtb_MultiportSwitch;

  /* MATLAB Function: '<S27>/engine massflow' incorporates:
   *  Gain: '<S27>/rpm2rad1'
   */
  Gen2_ref_enginemassflow(FILT_IN, Gen2_ref_B->T2s_filt.Switch,
    0.10471975511965977 * rtb_Switch13, rtb_etaVolConst_lt,
    Gen2_ref_B->BusInput3.eng.rVol_Hub_Eng, &Gen2_ref_B->sf_enginemassflow, inst);

  /* Switch: '<S27>/Switch' */
  if (Gen2_ref_B->BusInput3.bdcCbv.bFF_overspeed) {
    rtb_Switch2_a = rtb_DataTypeConversion15;
  } else {
    rtb_Switch2_a = rtb_Switch13;
  }

  /* End of Switch: '<S27>/Switch' */

  /* Switch: '<S114>/Switch2' incorporates:
   *  RelationalOperator: '<S114>/LowerRelop1'
   */
  if (!(rtb_DataTypeConversion15 > rtb_Switch2_a)) {
    /* Switch: '<S114>/Switch' incorporates:
     *  Constant: '<S27>/Constant4'
     *  RelationalOperator: '<S114>/UpperRelop'
     */
    if (rtb_DataTypeConversion15 < 1.0) {
      rtb_Switch2_a = 1.0;
    } else {
      rtb_Switch2_a = rtb_DataTypeConversion15;
    }

    /* End of Switch: '<S114>/Switch' */
  }

  /* End of Switch: '<S114>/Switch2' */

  /* MATLAB Function: '<S27>/engine massflow1' */
  u0 = 287.15 * Gen2_ref_B->T2s_filt.Switch;

  /* Switch: '<S27>/Switch1' incorporates:
   *  Saturate: '<S27>/Saturation4'
   */
  if (Gen2_ref_B->BusInput3.bdcCbv.bFF_low_boost) {
    delta_y = Gen2_ref_B->p2s_filt.Switch;
  } else if (Gen2_ref_B->p2s_filt.Switch <= 100000.0) {
    /* Saturate: '<S27>/Saturation4' */
    delta_y = 100000.0;
  } else {
    delta_y = Gen2_ref_B->p2s_filt.Switch;
  }

  /* End of Switch: '<S27>/Switch1' */

  /* MATLAB Function: '<S27>/engine massflow1' incorporates:
   *  Gain: '<S27>/rpm2rad'
   *  Product: '<S13>/Product1'
   */
  if (!(u0 >= 1.0)) {
    u0 = 1.0;
  }

  rtb_dm_e_tmp = rtb_etaVolConst_lt * Gen2_ref_B->BusInput3.eng.rVol_Hub_Eng;
  rtb_dm_e = rtb_dm_e_tmp * delta_y / u0 * (0.10471975511965977 * rtb_Switch2_a)
    / 2.0 / 6.2831853071795862;

  /* Gain: '<S27>/rpm2rad2' */
  rtb_Switch2_a = 1.0E-5 * FILT_IN;

  /* S-Function (sfix_look1_dyn): '<S27>/Lookup Table Dynamic1' */
  /* Dynamic Look-Up Table Block: '<S27>/Lookup Table Dynamic1'
   * Input0  Data Type:  Floating Point real_T
   * Input1  Data Type:  Floating Point real_T
   * Input2  Data Type:  Floating Point real_T
   * Output0 Data Type:  Floating Point real_T
   * Lookup Method: Linear_Endpoint
   *
   */
  LookUp_real_T_real_T( &(rtb_Divide2_f),
                       &Gen2_ref_B->BusInput3.bdcCbv.rRefCBVres_y[0],
                       rtb_Switch2_a, &Gen2_ref_B->
                       BusInput3.bdcCbv.rRefCBVres_x[0], 4U, inst);

  /* UnitDelay: '<S1>/Unit Delay' */
  FILT_IN = Gen2_ref_DWork->UnitDelay_DSTATE_i;

  /* Sum: '<S133>/Sum' */
  rtb_Switch2_a = rtb_Switch1_kk;

  /* RelationalOperator: '<S133>/Relational Operator' */
  rtb_LogicalOperator1_ix = (Gen2_ref_B->BusInput3.LR.rN_trig_cbv_lim <=
    rtb_Switch2_a);

  /* DiscreteIntegrator: '<S133>/Discrete-Time Integrator' */
  if (rtb_LogicalOperator1_ix ||
      (Gen2_ref_DWork->DiscreteTimeIntegrator_PrevR_no != 0)) {
    Gen2_ref_DWork->DiscreteTimeIntegrator_DSTATE_j = 0.0;
  }

  /* RelationalOperator: '<S133>/Relational Operator1' incorporates:
   *  DiscreteIntegrator: '<S133>/Discrete-Time Integrator'
   */
  rtb_RelationalOperator1_j = (Gen2_ref_B->BusInput3.LR.iNum_steady_state >
    Gen2_ref_DWork->DiscreteTimeIntegrator_DSTATE_j);

  /* Switch: '<S133>/Switch3' incorporates:
   *  Logic: '<S133>/Logical Operator4'
   */
  if (rtb_RelationalOperator1_j &&
      Gen2_ref_B->BusInput3.LR.bSwitch_Surge_CBV_Min) {
    /* S-Function (sfix_look1_dyn): '<S133>/Surge protection depending  on throttle position' */
    /* Dynamic Look-Up Table Block: '<S133>/Surge protection depending  on throttle position'
     * Input0  Data Type:  Floating Point real_T
     * Input1  Data Type:  Floating Point real_T
     * Input2  Data Type:  Floating Point real_T
     * Output0 Data Type:  Floating Point real_T
     * Lookup Method: Linear_Endpoint
     *
     */
    LookUp_real_T_real_T( &(rtb_Surgeprotectiondependingont),
                         &Gen2_ref_B->BusInput3.LR.rCBV_lim_byTV_Lup_y[0],
                         FILT_IN, &Gen2_ref_B->BusInput3.LR.rCBV_lim_byTV_Lup_x
                         [0], 4U, inst);
    FILT_IN = rtb_Surgeprotectiondependingont;
  } else {
    FILT_IN = Gen2_ref_B->BusInput3.bdcCbv.rPos_min;
  }

  /* End of Switch: '<S133>/Switch3' */

  /* Switch: '<S137>/Switch2' incorporates:
   *  RelationalOperator: '<S137>/LowerRelop1'
   *  RelationalOperator: '<S137>/UpperRelop'
   *  Switch: '<S137>/Switch'
   */
  if (FILT_IN > Gen2_ref_B->BusInput3.bdcCbv.rPos_max) {
    rtb_Switch2_a = Gen2_ref_B->BusInput3.bdcCbv.rPos_max;
  } else if (FILT_IN < Gen2_ref_B->BusInput3.bdcCbv.rPos_min) {
    /* Switch: '<S137>/Switch' */
    rtb_Switch2_a = Gen2_ref_B->BusInput3.bdcCbv.rPos_min;
  } else {
    rtb_Switch2_a = FILT_IN;
  }

  /* End of Switch: '<S137>/Switch2' */

  /* Switch: '<S1>/CBV Min' */
  if (rtb_LogicalOperator) {
    rtb_Switch1_kk = Gen2_ref_B->BusInput3.bdcCbv.rPos_min;
  } else {
    rtb_Switch1_kk = rtb_Switch2_a;
  }

  /* End of Switch: '<S1>/CBV Min' */

  /* Outputs for Atomic SubSystem: '<S27>/cbv tracking1' */
  /* Abs: '<S116>/Abs' */
  rtb_Abs_n = fabs(Gen2_ref_B->BusInput3.bdcCbv.rMaxErrCBVtracking);

  /* Logic: '<S116>/Logical Operator' incorporates:
   *  Logic: '<S116>/Logical Operator2'
   */
  rtb_LogicalOperator5_p = !Gen2_ref_B->BusInput3.bdcCbv.bFFonly_2nd_CBV;

  /* Logic: '<S116>/Logical Operator5' incorporates:
   *  Constant: '<S121>/Constant'
   *  Constant: '<S122>/Constant'
   *  DataTypeConversion: '<S1>/Data Type Conversion14'
   *  Logic: '<S116>/Logical Operator'
   *  Logic: '<S116>/Logical Operator1'
   *  Logic: '<S116>/Logical Operator2'
   *  Logic: '<S116>/Logical Operator3'
   *  Logic: '<S116>/Logical Operator4'
   *  Logic: '<S116>/Logical Operator6'
   *  Logic: '<S1>/Logical Operator5'
   *  RelationalOperator: '<S121>/Compare'
   *  RelationalOperator: '<S122>/Compare'
   */
  rtb_LogicalOperator5_p = ((((!(Gen2_ref_B->BusInput3.eng.rNum_CBV > 1.5)) ||
    rtb_LogicalOperator5_p) && ((!(Gen2_ref_B->BusInput3.eng.rNum_CBV > 2.5)) ||
    (rtb_LogicalOperator5_p && (!Gen2_ref_B->BusInput3.bdcCbv.bFFonly_3rd_CBV))))
    || (!Gen2_ref_B->BusInput3.bdcCbv.bCBVtracking2nd3rdCBV) || (!(rtb_Sum1_dh
    != 0.0)));

  /* DiscreteIntegrator: '<S116>/Discrete-Time Integrator' */
  if (rtb_LogicalOperator5_p || (Gen2_ref_DWork->DiscreteTimeIntegrator_PrevR_lh
       != 0)) {
    Gen2_ref_DWork->DiscreteTimeIntegrator_DSTAT_iq = 0.0;
  }

  r = Gen2_ref_DWork->DiscreteTimeIntegrator_DSTAT_iq;

  /* End of DiscreteIntegrator: '<S116>/Discrete-Time Integrator' */

  /* Switch: '<S116>/Switch8' incorporates:
   *  Constant: '<S116>/max_PR1'
   */
  if (Gen2_ref_B->TON2.LogicalOperator3) {
    /* Sum: '<S116>/Sum' incorporates:
     *  UnitDelay: '<S1>/Unit Delay5'
     */
    rtb_Sum_mf = Gen2_ref_DWork->UnitDelay5_DSTATE -
      Gen2_ref_B->BusInput3.bdcCbv.rRefCBVtracking;

    /* Switch: '<S116>/Switch4' incorporates:
     *  Constant: '<S116>/max_PR5'
     *  Constant: '<S116>/max_PR6'
     *  RelationalOperator: '<S116>/Relational Operator3'
     *  Sum: '<S116>/Sum5'
     *  UnitDelay: '<S27>/Unit Delay6'
     */
    if (Gen2_ref_DWork->UnitDelay6_DSTATE >
        Gen2_ref_B->BusInput3.bdcCbv.rPos_max - 0.001) {
      FILT_IN = 0.0;
    } else {
      FILT_IN = rtb_Abs_n;
    }

    /* End of Switch: '<S116>/Switch4' */

    /* Switch: '<S123>/Switch2' incorporates:
     *  RelationalOperator: '<S123>/LowerRelop1'
     */
    if (!(rtb_Sum_mf > FILT_IN)) {
      /* Switch: '<S116>/Switch5' incorporates:
       *  Constant: '<S116>/max_PR5'
       *  Constant: '<S116>/max_PR6'
       *  Gain: '<S116>/Gain2'
       *  RelationalOperator: '<S116>/Relational Operator2'
       *  Sum: '<S116>/Sum4'
       *  UnitDelay: '<S27>/Unit Delay6'
       */
      if (Gen2_ref_DWork->UnitDelay6_DSTATE < rtb_Switch1_kk + 0.001) {
        FILT_IN = 0.0;
      } else {
        FILT_IN = -rtb_Abs_n;
      }

      /* End of Switch: '<S116>/Switch5' */

      /* Switch: '<S123>/Switch' incorporates:
       *  RelationalOperator: '<S123>/UpperRelop'
       */
      if (!(rtb_Sum_mf < FILT_IN)) {
        FILT_IN = rtb_Sum_mf;
      }

      /* End of Switch: '<S123>/Switch' */
    }

    /* End of Switch: '<S123>/Switch2' */
  } else {
    FILT_IN = 0.0;
  }

  /* End of Switch: '<S116>/Switch8' */

  /* Update for DiscreteIntegrator: '<S116>/Discrete-Time Integrator' incorporates:
   *  Product: '<S116>/Divide'
   */
  Gen2_ref_DWork->DiscreteTimeIntegrator_DSTAT_iq +=
    Gen2_ref_B->BusInput3.bdcCbv.rKiCBVtracking * FILT_IN * 0.01;
  Gen2_ref_DWork->DiscreteTimeIntegrator_PrevR_lh = (int8_T)
    rtb_LogicalOperator5_p;

  /* End of Outputs for SubSystem: '<S27>/cbv tracking1' */

  /* Sum: '<S27>/Sum3' incorporates:
   *  Constant: '<S27>/Constant'
   *  Sum: '<S27>/Sum5'
   */
  FILT_IN = (rtb_Divide2_f + r) + 1.0;

  /* MultiPortSwitch: '<S25>/Multiport Switch1' incorporates:
   *  BusCreator: '<S23>/Bus Creator1'
   */
  if ((int32_T)Gen2_ref_B->sf_MATLABFunction_e.y == 1) {
    rtb_Divide2_f = Gen2_ref_B->Filter1.Switch1;
  } else {
    rtb_Divide2_f = Gen2_ref_B->Filter4.Switch1;
  }

  /* End of MultiPortSwitch: '<S25>/Multiport Switch1' */

  /* Gain: '<S1>/Gain1' */
  r = 100000.0 * rtb_Divide2_f;

  /* DataTypeConversion: '<S117>/Data Type Conversion' */
  rtb_Divide2_f = Gen2_ref_B->BusInput3.bdcCbv.bDynFFcbv_ON;

  /* Sum: '<S117>/Sum3' incorporates:
   *  Sum: '<S175>/Sum3'
   */
  rtb_Saturation_cx = Gen2_ref_B->BusInput3.eng.rVol_IC_HP +
    Gen2_ref_B->BusInput3.eng.rVol_IC_LP;
  rtb_Sum_mf = rtb_Saturation_cx;

  /* Product: '<S117>/Divide6' incorporates:
   *  Constant: '<S117>/R_air'
   *  Product: '<S117>/Divide7'
   */
  rtb_Abs_n = rtb_Sum_mf / (287.15 * Gen2_ref_B->T2s_filt.Switch);

  /* Saturate: '<S27>/Saturation5' */
  if (Gen2_ref_B->BusInput3.eng.rNum_CBV > 10.0) {
    rtb_Sum_mf = 10.0;
  } else if (Gen2_ref_B->BusInput3.eng.rNum_CBV < 1.0) {
    rtb_Sum_mf = 1.0;
  } else {
    rtb_Sum_mf = Gen2_ref_B->BusInput3.eng.rNum_CBV;
  }

  /* End of Saturate: '<S27>/Saturation5' */

  /* Product: '<S27>/Divide1' incorporates:
   *  Product: '<S117>/Divide8'
   *  Product: '<S27>/Product'
   *  Sum: '<S27>/Sum1'
   *  Sum: '<S27>/Sum2'
   */
  rtb_Sum_mf = ((rtb_dm_e * FILT_IN - r * rtb_Divide2_f * rtb_Abs_n) -
                Gen2_ref_B->sf_enginemassflow.dm_e) / rtb_Sum_mf;

  /* Saturate: '<S27>/Saturation' */
  if (rtb_Sum_mf <= 0.0) {
    rtb_Abs_n = 0.0;
  } else {
    rtb_Abs_n = rtb_Sum_mf;
  }

  /* End of Saturate: '<S27>/Saturation' */

  /* MultiPortSwitch: '<S25>/Multiport Switch2' incorporates:
   *  BusCreator: '<S23>/Bus Creator1'
   */
  if ((int32_T)Gen2_ref_B->sf_MATLABFunction_e.y == 1) {
    FILT_IN = rtb_Switch2_h1;
  } else {
    FILT_IN = rtb_BusCreator1_ref_P2_FF;
  }

  /* End of MultiPortSwitch: '<S25>/Multiport Switch2' */

  /* Switch: '<S106>/Switch2' incorporates:
   *  Constant: '<S25>/Constant'
   *  RelationalOperator: '<S106>/LowerRelop1'
   */
  if (FILT_IN > 1.0E+6) {
    rtb_Sum_mf = 1.0E+6;
  } else {
    /* Gain: '<S25>/Gain1' */
    r = rtb_kW2W1_h;

    /* S-Function (sfix_look1_dyn): '<S25>/Lookup Table Dynamic' */
    /* Dynamic Look-Up Table Block: '<S25>/Lookup Table Dynamic'
     * Input0  Data Type:  Floating Point real_T
     * Input1  Data Type:  Floating Point real_T
     * Input2  Data Type:  Floating Point real_T
     * Output0 Data Type:  Floating Point real_T
     * Lookup Method: Linear_Endpoint
     *
     */
    LookUp_real_T_real_T( &(rtb_Sum1_lo),
                         &Gen2_ref_B->BusInput3.traj.rPrR_deltaP_TV_y[0], r,
                         &rtb_Gain1_eu[0], 4U, inst);

    /* Sum: '<S25>/Sum1' incorporates:
     *  Product: '<S25>/Product2'
     */
    rtb_Sum1_lo = rtb_Sum1_lo * rtb_Saturation1_i + rtb_MultiportSwitch;

    /* Switch: '<S106>/Switch' incorporates:
     *  RelationalOperator: '<S106>/UpperRelop'
     */
    if (FILT_IN < rtb_Sum1_lo) {
      rtb_Sum_mf = rtb_Sum1_lo;
    } else {
      rtb_Sum_mf = FILT_IN;
    }

    /* End of Switch: '<S106>/Switch' */
  }

  /* Gain: '<S1>/Gain2' */
  rtb_Sum1_lo = 100000.0 * rtb_Sum_mf;

  /* MATLAB Function: '<S27>/MATLAB Function1' incorporates:
   *  Constant: '<S1>/Constant2'
   *  Constant: '<S27>/Constant3'
   *  Product: '<S27>/Product1'
   */
  if (rtb_Sum1_lo >= 100000.0) {
    r = 100000.0 / rtb_Sum1_lo;
    if (1.0E-6 >= r) {
      r = 1.0E-6;
    }

    if (1.0 / r <= 1.8929291587378541) {
      u0 = 0.78539816339744828 * Gen2_ref_B->BusInput3.bdcCbv.rDref *
        Gen2_ref_B->BusInput3.bdcCbv.rDref * rtb_Sum1_lo / sqrt(287.15 *
        Gen2_ref_B->T2s_filt.Switch) * sqrt((rt_powd_snf(r, 1.4285714285714286, inst)
        - rt_powd_snf(r, 1.7142857142857144, inst)) * 7.0000000000000009);
      if (!(u0 >= 1.0E-6)) {
        u0 = 1.0E-6;
      }

      rtb_Sum1_lo = rtb_Abs_n / u0;
    } else {
      u0 = 0.78539816339744828 * Gen2_ref_B->BusInput3.bdcCbv.rDref *
        Gen2_ref_B->BusInput3.bdcCbv.rDref * rtb_Sum1_lo / sqrt(287.15 *
        Gen2_ref_B->T2s_filt.Switch) * 0.6847314563772704;
      if (!(u0 >= 1.0E-6)) {
        u0 = 1.0E-6;
      }

      rtb_Sum1_lo = rtb_Abs_n / u0;
    }
  } else {
    rtb_Sum1_lo = 0.0;
  }

  /* End of MATLAB Function: '<S27>/MATLAB Function1' */

  /* Saturate: '<S27>/Saturation1' */
  if (rtb_Sum1_lo > 1.0) {
    rtb_Sum_mf = 1.0;
  } else if (rtb_Sum1_lo < 0.0) {
    rtb_Sum_mf = 0.0;
  } else {
    rtb_Sum_mf = rtb_Sum1_lo;
  }

  /* End of Saturate: '<S27>/Saturation1' */

  /* S-Function (sfix_look1_dyn): '<S27>/Lookup Table Dynamic' */
  /* Dynamic Look-Up Table Block: '<S27>/Lookup Table Dynamic'
   * Input0  Data Type:  Floating Point real_T
   * Input1  Data Type:  Floating Point real_T
   * Input2  Data Type:  Floating Point real_T
   * Output0 Data Type:  Floating Point real_T
   * Lookup Method: Linear_Endpoint
   *
   */
  LookUp_real_T_real_T( &(rtb_Divide2_f),
                       &Gen2_ref_B->BusInput3.bdcCbv.rCd_vect_x[0], rtb_Sum_mf,
                       &Gen2_ref_B->BusInput3.bdcCbv.rCd_vect_y[0], 10U, inst);

  /* MinMax: '<S27>/MinMax' */
  r = Gen2_ref_B->BusInput3.bdcCbv.rCd_vect_x[0];
  for (k = 0; k < 10; k++) {
    u1 = Gen2_ref_B->BusInput3.bdcCbv.rCd_vect_x[k + 1];
    if ((!(r >= u1)) && (!rtIsNaN(u1))) {
      r = u1;
    }
  }

  /* End of MinMax: '<S27>/MinMax' */

  /* Abs: '<S112>/Abs' */
  FILT_IN = fabs(r);

  /* Switch: '<S112>/Switch' incorporates:
   *  Constant: '<S112>/Constant2'
   *  RelationalOperator: '<S112>/Relational Operator'
   */
  if (2.2204460492503131E-16 >= FILT_IN) {
    r = 2.2204460492503131E-16;
  }

  /* End of Switch: '<S112>/Switch' */

  /* Product: '<S27>/Divide' */
  delta_y = rtb_Divide2_f / r;
  for (i = 0; i < 5; i++) {
    /* Gain: '<S27>/Gain1' */
    rtb_Gain1_eu[i] = 0.01 * Gen2_ref_B->BusInput3.bdcCbv.rRefCBVconvert_x[i];

    /* Gain: '<S27>/Gain2' */
    rtb_Gain2_k[i] = 0.01 * Gen2_ref_B->BusInput3.bdcCbv.rRefCBVconvert_y[i];
  }

  /* S-Function (sfix_look1_dyn): '<S27>/Lookup Table Dynamic2' */
  /* Dynamic Look-Up Table Block: '<S27>/Lookup Table Dynamic2'
   * Input0  Data Type:  Floating Point real_T
   * Input1  Data Type:  Floating Point real_T
   * Input2  Data Type:  Floating Point real_T
   * Output0 Data Type:  Floating Point real_T
   * Lookup Method: Linear_Endpoint
   *
   */
  LookUp_real_T_real_T( &(FILT_IN), &rtb_Gain2_k[0], delta_y, &rtb_Gain1_eu[0],
                       4U, inst);

  /* Saturate: '<S27>/Saturation3' */
  if (Gen2_ref_B->BusInput3.eng.rNum_CBV > 1.0) {
    r = 1.0;
  } else if (Gen2_ref_B->BusInput3.eng.rNum_CBV < 0.0) {
    r = 0.0;
  } else {
    r = Gen2_ref_B->BusInput3.eng.rNum_CBV;
  }

  /* End of Saturate: '<S27>/Saturation3' */

  /* Product: '<S27>/Divide2' */
  rtb_Divide2_f = FILT_IN * r;

  /* Switch: '<S115>/Switch2' incorporates:
   *  RelationalOperator: '<S115>/LowerRelop1'
   *  RelationalOperator: '<S115>/UpperRelop'
   *  Switch: '<S115>/Switch'
   */
  if (rtb_Divide2_f > Gen2_ref_B->BusInput3.bdcCbv.rPos_max) {
    rtb_Sum1_lo = Gen2_ref_B->BusInput3.bdcCbv.rPos_max;
  } else if (rtb_Divide2_f < rtb_Switch1_kk) {
    /* Switch: '<S115>/Switch' */
    rtb_Sum1_lo = rtb_Switch1_kk;
  } else {
    rtb_Sum1_lo = rtb_Divide2_f;
  }

  /* End of Switch: '<S115>/Switch2' */

  /* Switch: '<S26>/Switch4' incorporates:
   *  Constant: '<S26>/Constant1'
   */
  if (Gen2_ref_B->BusInput3.bdcCbv.bActive_ff) {
    FILT_IN = rtb_Sum1_lo;
  } else {
    FILT_IN = 0.0;
  }

  /* End of Switch: '<S26>/Switch4' */

  /* Saturate: '<S26>/Saturation1' */
  if (FILT_IN > 1.0) {
    rtb_Saturation1_i = 1.0;
  } else if (FILT_IN < 0.0) {
    rtb_Saturation1_i = 0.0;
  } else {
    rtb_Saturation1_i = FILT_IN;
  }

  /* End of Saturate: '<S26>/Saturation1' */

  /* Switch: '<S41>/Switch2' incorporates:
   *  Sum: '<S41>/Sum'
   *  Sum: '<S41>/Sum7'
   */
  if (rtb_LogicalOperator) {
    /* S-Function (sfix_look1_dyn): '<S41>/Lookup4' */
    /* Dynamic Look-Up Table Block: '<S41>/Lookup4'
     * Input0  Data Type:  Floating Point real_T
     * Input1  Data Type:  Floating Point real_T
     * Input2  Data Type:  Floating Point real_T
     * Output0 Data Type:  Floating Point real_T
     * Lookup Method: Linear_Endpoint
     *
     */
    LookUp_real_T_real_T( &(rtb_Lookup4), &Gen2_ref_B->BusInput3.bdcCbv.rKp_Lup
                         [0], rtb_Pa2bar,
                         &Gen2_ref_B->BusInput3.bdcMisc.rPr_Lup_in[0], 9U, inst);
    FILT_IN = rtb_Lookup4 + Gen2_ref_B->BusInput3.bdcCbv.rKp_grid_offset;
  } else {
    /* S-Function (sfix_look1_dyn): '<S41>/Lookup5' */
    /* Dynamic Look-Up Table Block: '<S41>/Lookup5'
     * Input0  Data Type:  Floating Point real_T
     * Input1  Data Type:  Floating Point real_T
     * Input2  Data Type:  Floating Point real_T
     * Output0 Data Type:  Floating Point real_T
     * Lookup Method: Linear_Endpoint
     *
     */
    LookUp_real_T_real_T( &(rtb_Lookup5),
                         &Gen2_ref_B->BusInput3.bdcCbv.rKp_island_Lup[0],
                         rtb_Pa2bar, &Gen2_ref_B->BusInput3.bdcMisc.rPr_Lup_in[0],
                         9U, inst);
    FILT_IN = rtb_Lookup5 + Gen2_ref_B->BusInput3.bdcCbv.rKp_island_offset;
  }

  /* End of Switch: '<S41>/Switch2' */

  /* S-Function (sfix_look1_dyn): '<S41>/Lookup9' */
  /* Dynamic Look-Up Table Block: '<S41>/Lookup9'
   * Input0  Data Type:  Floating Point real_T
   * Input1  Data Type:  Floating Point real_T
   * Input2  Data Type:  Floating Point real_T
   * Output0 Data Type:  Floating Point real_T
   * Lookup Method: Linear_Endpoint
   *
   */
  LookUp_real_T_real_T( &(r), &Gen2_ref_B->BusInput3.bdcCbv.rGainMultRej_y[0],
                       rtb_DataTypeConversion15,
                       &Gen2_ref_B->BusInput3.bdcCbv.rGainMultRej_x[0], 4U, inst);

  /* Product: '<S41>/Product1' */
  rtb_Divide2_f = FILT_IN * r;

  /* Switch: '<S130>/Switch2' incorporates:
   *  RelationalOperator: '<S130>/LowerRelop1'
   *  RelationalOperator: '<S130>/UpperRelop'
   *  Switch: '<S130>/Switch'
   */
  if (rtb_Divide2_f > Gen2_ref_B->BusInput3.bdcMisc.rKpMax) {
    rtb_Divide2_f = Gen2_ref_B->BusInput3.bdcMisc.rKpMax;
  } else if (rtb_Divide2_f < Gen2_ref_B->BusInput3.bdcMisc.rKpMin) {
    /* Switch: '<S130>/Switch' */
    rtb_Divide2_f = Gen2_ref_B->BusInput3.bdcMisc.rKpMin;
  }

  /* End of Switch: '<S130>/Switch2' */

  /* Logic: '<S1>/Logical Operator3' incorporates:
   *  DataTypeConversion: '<S1>/Data Type Conversion13'
   */
  rtb_LogicalOperator5_p = !(rtb_Sum1_dh != 0.0);

  /* MATLAB Function: '<S26>/fb_err' incorporates:
   *  BusCreator: '<S23>/Bus Creator1'
   *  SignalConversion generated from: '<S110>/ SFunction '
   */
  if ((!Gen2_ref_DWork->err_1_not_empty_d) || rtb_LogicalOperator5_p) {
    Gen2_ref_DWork->err_1_a = 0.0;
    Gen2_ref_DWork->err_1_not_empty_d = true;
  }

  err = rtb_Divide2 * rtb_Divide1_fn - rtb_BusCreator1_ref_P2_FB_CBV;
  FILT_IN = Gen2_ref_DWork->err_1_a - err;
  Gen2_ref_DWork->err_1_a = err;

  /* Product: '<S26>/Product' incorporates:
   *  MATLAB Function: '<S26>/fb_err'
   */
  rtb_up = rtb_Divide2_f * err;

  /* Logic: '<S26>/Logical Operator1' incorporates:
   *  Logic: '<S26>/Logical Operator2'
   *  RelationalOperator: '<S107>/FixPt Relational Operator'
   *  UnitDelay: '<S107>/Delay Input1'
   */
  rtb_bCBV_min = ((Gen2_ref_B->BusInput3.bdcCbv.bActive_ff !=
                   Gen2_ref_DWork->DelayInput1_DSTATE_fv) &&
                  ((!rtb_LogicalOperator5_p) && rtb_LogicalOperator_b));

  /* Logic: '<S26>/Logical Operator' incorporates:
   *  MATLAB Function: '<S26>/fb_err'
   */
  rtb_LogicalOperator_b = (Gen2_ref_B->BusInput.tLvrt.bLvrtFlg ||
    rtb_LogicalOperator5_p || rtb_bCBV_min);

  /* Delay: '<S26>/Delay' */
  if (Gen2_ref_DWork->icLoad_kq) {
    Gen2_ref_DWork->Delay_DSTATE_hq = rtb_Saturation1_i;
  }

  /* Sum: '<S111>/Add2' */
  rtb_Add2_h = (Gen2_ref_B->BusInput3.bdcCbv.rPos_Start - rtb_Saturation1_i) -
    rtb_up;

  /* Delay: '<S111>/Delay' */
  if ((((Gen2_ref_PrevZCSigState->Delay_Reset_ZCE_kk == 1) != (int32_T)
        rtb_LogicalOperator5_p) && (Gen2_ref_PrevZCSigState->Delay_Reset_ZCE_kk
        != 3)) || rtb_LogicalOperator5_p) {
    Gen2_ref_DWork->Delay_DSTATE_ow = 0.0;
  }

  Gen2_ref_PrevZCSigState->Delay_Reset_ZCE_kk = rtb_LogicalOperator5_p;

  /* Switch: '<S26>/Switch1' incorporates:
   *  Delay: '<S111>/Delay2'
   *  Delay: '<S26>/Delay'
   *  Sum: '<S26>/Sum'
   *  Sum: '<S26>/Sum3'
   *  Switch: '<S111>/Switch3'
   *  UnitDelay: '<S26>/Unit Delay1'
   */
  if (rtb_bCBV_min) {
    rtb_Add2_h = (Gen2_ref_DWork->Delay_DSTATE_hq - rtb_Saturation1_i) +
      Gen2_ref_DWork->UnitDelay1_DSTATE_c;
  } else if (!Gen2_ref_DWork->Delay2_DSTATE_k) {
    /* Switch: '<S111>/Switch1' incorporates:
     *  Delay: '<S111>/Delay'
     *  Product: '<S26>/Product3'
     *  Sum: '<S111>/Add1'
     *  Sum: '<S111>/Add3'
     *  Switch: '<S111>/Switch'
     *  Switch: '<S111>/Switch3'
     */
    if (Gen2_ref_B->BusInput.tLvrt.bLvrtFlg) {
      rtb_Add2_h = (Gen2_ref_B->BusInput.tLvrt.rCbvPosFb - rtb_Saturation1_i) -
        rtb_up;
    } else {
      if (!rtb_LogicalOperator5_p) {
        /* Switch: '<S111>/Switch' incorporates:
         *  Constant: '<S111>/Constant'
         */
        rtb_Add2_h = 0.0;
      }

      rtb_Add2_h = (FILT_IN * rtb_Divide2_f + rtb_Add2_h) +
        Gen2_ref_DWork->Delay_DSTATE_ow;
    }

    /* End of Switch: '<S111>/Switch1' */
  }

  /* End of Switch: '<S26>/Switch1' */

  /* DiscreteIntegrator: '<S26>/Discrete-Time Integrator' */
  if (Gen2_ref_DWork->DiscreteTimeIntegrator_IC_LOA_l != 0) {
    Gen2_ref_DWork->DiscreteTimeIntegrator_DSTAT_ja = rtb_Add2_h;
  }

  if (rtb_LogicalOperator_b || (Gen2_ref_DWork->DiscreteTimeIntegrator_PrevRe_c
       != 0)) {
    Gen2_ref_DWork->DiscreteTimeIntegrator_DSTAT_ja = rtb_Add2_h;
  }

  rtb_MultiportSwitch = Gen2_ref_DWork->DiscreteTimeIntegrator_DSTAT_ja;

  /* Switch: '<S26>/Switch6' incorporates:
   *  Constant: '<S26>/Constant5'
   *  DiscreteIntegrator: '<S26>/Discrete-Time Integrator'
   *  Sum: '<S26>/Sum1'
   */
  if (Gen2_ref_B->BusInput3.bdcCbv.bFFonly) {
    FILT_IN = 0.0;
  } else {
    FILT_IN = rtb_up + Gen2_ref_DWork->DiscreteTimeIntegrator_DSTAT_ja;
  }

  /* End of Switch: '<S26>/Switch6' */

  /* BusCreator: '<Root>/Bus Creator' incorporates:
   *  BusCreator: '<S26>/Bus Creator1'
   *  DataTypeConversion: '<S26>/Data Type Conversion1'
   *  Outport: '<Root>/dbg'
   */
  Gen2_ref_Y->dbg.BDC.cbv.fb_cbv = (real32_T)FILT_IN;

  /* Sum: '<S26>/Sum5' */
  r = rtb_Saturation1_i + FILT_IN;

  /* Gain: '<S427>/Gain5' */
  FILT_IN = 0.001 * Gen2_ref_B->BusInput3.LR.rTi_LR_ActSat_CBV;

  /* Outputs for Atomic SubSystem: '<S427>/TP_ActSat_CBV' */
  /* Logic: '<S427>/Logical Operator1' incorporates:
   *  Bias: '<S427>/ u+Ts6'
   *  Delay: '<S427>/Delay'
   *  RelationalOperator: '<S427>/Relational Operator15'
   *  RelationalOperator: '<S427>/Relational Operator18'
   */
  Gen2_ref_TP_ActSat_CBV((rtb_RelationalOperator2_j &&
    Gen2_ref_B->BusInput3.LR.bP_LoadReject_Active &&
    (Gen2_ref_DWork->Delay_DSTATE[0] >=
     Gen2_ref_B->BusInput3.LR.rP_LR_Trig_ActSat_CBV) && (rtb_Saturation >
    Gen2_ref_B->BusInput3.LR.rP_LR_Trig_ActSat_CBV) &&
    Gen2_ref_B->BusInput3.LR.bLR_ActSat_CBV), FILT_IN + 0.01,
    &Gen2_ref_B->TP_ActSat_CBV, &Gen2_ref_DWork->TP_ActSat_CBV, inst);

  /* End of Outputs for SubSystem: '<S427>/TP_ActSat_CBV' */

  /* Switch: '<S26>/Switch2' incorporates:
   *  MinMax: '<S26>/MinMax'
   *  RelationalOperator: '<S108>/LowerRelop1'
   *  Switch: '<S108>/Switch2'
   */
  if (Gen2_ref_B->TP_ActSat_CBV.LogicalOperator1) {
    rtb_Switch1_kk = Gen2_ref_B->BusInput3.bdcCbv.rPos_max;
  } else if (r > Gen2_ref_B->BusInput3.bdcCbv.rPos_max) {
    /* Switch: '<S108>/Switch2' */
    rtb_Switch1_kk = Gen2_ref_B->BusInput3.bdcCbv.rPos_max;
  } else {
    if ((rtb_Switch1_kk >= Gen2_ref_B->BusInput3.bdcCbv.rPos_min) || rtIsNaN
        (Gen2_ref_B->BusInput3.bdcCbv.rPos_min)) {
      /* MinMax: '<S26>/MinMax' incorporates:
       *  Switch: '<S108>/Switch2'
       */
      FILT_IN = rtb_Switch1_kk;
    } else {
      /* MinMax: '<S26>/MinMax' incorporates:
       *  Switch: '<S108>/Switch2'
       */
      FILT_IN = Gen2_ref_B->BusInput3.bdcCbv.rPos_min;
    }

    /* Switch: '<S108>/Switch' incorporates:
     *  RelationalOperator: '<S108>/UpperRelop'
     *  Switch: '<S108>/Switch2'
     */
    if (r < FILT_IN) {
      rtb_Switch1_kk = FILT_IN;
    } else {
      rtb_Switch1_kk = r;
    }

    /* End of Switch: '<S108>/Switch' */
  }

  /* End of Switch: '<S26>/Switch2' */

  /* Switch: '<S41>/Switch3' incorporates:
   *  Sum: '<S41>/Sum1'
   *  Sum: '<S41>/Sum6'
   */
  if (rtb_LogicalOperator) {
    /* S-Function (sfix_look1_dyn): '<S41>/Lookup6' */
    /* Dynamic Look-Up Table Block: '<S41>/Lookup6'
     * Input0  Data Type:  Floating Point real_T
     * Input1  Data Type:  Floating Point real_T
     * Input2  Data Type:  Floating Point real_T
     * Output0 Data Type:  Floating Point real_T
     * Lookup Method: Linear_Endpoint
     *
     */
    LookUp_real_T_real_T( &(rtb_Lookup6), &Gen2_ref_B->BusInput3.bdcCbv.rKi_Lup
                         [0], rtb_Pa2bar,
                         &Gen2_ref_B->BusInput3.bdcMisc.rPr_Lup_in[0], 9U, inst);
    FILT_IN = rtb_Lookup6 + Gen2_ref_B->BusInput3.bdcCbv.rKi_grid_offset;
  } else {
    /* Logic: '<S41>/Logical Operator' */
    rtb_bCBV_min = (rtb_Switch4_j &&
                    Gen2_ref_B->BusInput3.bdcCbv.bKi_island_reject);

    /* Switch: '<S41>/Switch5' */
    for (i = 0; i < 10; i++) {
      if (rtb_bCBV_min) {
        rtb_Switch6_n[i] = Gen2_ref_B->BusInput3.bdcCbv.rKi_island_reject_Lup[i];
      } else {
        rtb_Switch6_n[i] = Gen2_ref_B->BusInput3.bdcCbv.rKi_island_Lup[i];
      }
    }

    /* End of Switch: '<S41>/Switch5' */

    /* S-Function (sfix_look1_dyn): '<S41>/Lookup7' */
    /* Dynamic Look-Up Table Block: '<S41>/Lookup7'
     * Input0  Data Type:  Floating Point real_T
     * Input1  Data Type:  Floating Point real_T
     * Input2  Data Type:  Floating Point real_T
     * Output0 Data Type:  Floating Point real_T
     * Lookup Method: Linear_Endpoint
     *
     */
    LookUp_real_T_real_T( &(rtb_Lookup7), &rtb_Switch6_n[0], rtb_Pa2bar,
                         &Gen2_ref_B->BusInput3.bdcMisc.rPr_Lup_in[0], 9U, inst);
    FILT_IN = rtb_Lookup7 + Gen2_ref_B->BusInput3.bdcCbv.rKi_island_offset;
  }

  /* End of Switch: '<S41>/Switch3' */

  /* Switch: '<S131>/Switch2' incorporates:
   *  RelationalOperator: '<S131>/LowerRelop1'
   *  RelationalOperator: '<S131>/UpperRelop'
   *  Switch: '<S131>/Switch'
   */
  if (FILT_IN > Gen2_ref_B->BusInput3.bdcMisc.rKiMax) {
    rtb_Pa2bar = Gen2_ref_B->BusInput3.bdcMisc.rKiMax;
  } else if (FILT_IN < Gen2_ref_B->BusInput3.bdcMisc.rKiMin) {
    /* Switch: '<S131>/Switch' */
    rtb_Pa2bar = Gen2_ref_B->BusInput3.bdcMisc.rKiMin;
  } else {
    rtb_Pa2bar = FILT_IN;
  }

  /* End of Switch: '<S131>/Switch2' */

  /* Switch: '<S26>/Switch5' incorporates:
   *  Constant: '<S26>/Constant4'
   *  Product: '<S26>/Divide'
   *  RelationalOperator: '<S26>/Relational Operator'
   */
  if (Gen2_ref_B->BusInput3.bdcCbv.rKaw <= 0.0) {
    /* Saturate: '<S26>/Saturation' */
    if (rtb_Divide2_f <= 0.1) {
      rtb_Divide2_f = 0.1;
    }

    /* End of Saturate: '<S26>/Saturation' */
    FILT_IN = rtb_Pa2bar / rtb_Divide2_f;
  } else {
    FILT_IN = Gen2_ref_B->BusInput3.bdcCbv.rKaw;
  }

  /* End of Switch: '<S26>/Switch5' */

  /* Product: '<S26>/Product2' incorporates:
   *  Sum: '<S26>/Sum4'
   */
  rtb_Divide2_f = (rtb_Switch1_kk - r) * FILT_IN;

  /* Switch: '<S109>/Switch2' incorporates:
   *  Constant: '<S26>/Constant2'
   *  RelationalOperator: '<S109>/LowerRelop1'
   *  RelationalOperator: '<S109>/UpperRelop'
   *  Switch: '<S109>/Switch'
   */
  if (rtb_Divide2_f > 1.0E+10) {
    FILT_IN = 1.0E+10;
  } else if (rtb_Divide2_f < Gen2_ref_B->BusInput3.bdcCbv.rAW_lim_rej) {
    /* Switch: '<S109>/Switch' */
    FILT_IN = Gen2_ref_B->BusInput3.bdcCbv.rAW_lim_rej;
  } else {
    FILT_IN = rtb_Divide2_f;
  }

  /* End of Switch: '<S109>/Switch2' */

  /* BusCreator: '<Root>/Bus Creator' incorporates:
   *  BusCreator: '<S43>/Bus Creator6'
   *  DataTypeConversion: '<S43>/Data Type Conversion2'
   *  DataTypeConversion: '<S43>/Data Type Conversion4'
   *  Outport: '<Root>/dbg'
   */
  Gen2_ref_Y->dbg.BDC.SP.rMdot_mixture_Bypass = (real32_T)x;
  Gen2_ref_Y->dbg.BDC.SP.mdot_corr = (real32_T)rtb_Switch_n;

  /* Sum: '<S23>/Sum6' */
  rtb_Divide2_f = rtb_Sum_c - rtb_Gain_kl;

  /* Product: '<S62>/Product' incorporates:
   *  MATLAB Function: '<S62>/MATLAB Function'
   */
  rtb_Sum_c = (rtb_LogicalOperator2_ov ? (real_T)Gen2_ref_DWork->x_i : 0.0) *
    rtb_Divide2_f;

  /* Outputs for Atomic SubSystem: '<S62>/Filter3' */
  Gen2_ref_Filter3(rtb_Sum_c, Gen2_ref_B->BusInput3.traj.rTiFp2sComp,
                   Gen2_ref_ConstB.Constant11, rtb_LogicalOperator2_dc,
                   &Gen2_ref_B->Filter3, &Gen2_ref_DWork->Filter3, inst);

  /* End of Outputs for SubSystem: '<S62>/Filter3' */

  /* Switch: '<S62>/Switch4' incorporates:
   *  DiscreteIntegrator: '<S62>/Discrete-Time Integrator'
   *  Gain: '<S62>/Gain6'
   *  Product: '<S62>/Divide'
   *  Product: '<S62>/Product3'
   *  Switch: '<S62>/Switch'
   */
  if (rtb_LogicalOperator_aw) {
    /* Switch: '<S96>/Switch' incorporates:
     *  Abs: '<S96>/Abs'
     *  Constant: '<S96>/Constant2'
     *  RelationalOperator: '<S96>/Relational Operator'
     */
    if (2.2204460492503131E-16 >= fabs(Gen2_ref_B->BusInput3.traj.rTiFp2sComp))
    {
      delta_y = 2.2204460492503131E-16;
    } else {
      delta_y = Gen2_ref_B->BusInput3.traj.rTiFp2sComp;
    }

    /* End of Switch: '<S96>/Switch' */
    rtb_Gain_kl = -Gen2_ref_DWork->DiscreteTimeIntegrator_DSTATE_a / delta_y;
  } else {
    if (!Gen2_ref_B->BusInput3.traj.bUseUnFilterComp) {
      /* Switch: '<S62>/Switch' */
      rtb_Sum_c = Gen2_ref_B->Filter3.Switch;
    }

    /* Switch: '<S62>/Switch2' incorporates:
     *  Abs: '<S62>/Abs2'
     *  Constant: '<S62>/Constant2'
     *  Logic: '<S62>/Logical Operator3'
     *  Logic: '<S62>/Logical Operator7'
     *  Logic: '<S62>/Logical Operator8'
     *  MATLAB Function: '<S62>/MATLAB Function'
     *  RelationalOperator: '<S62>/Relational Operator4'
     *  RelationalOperator: '<S62>/Relational Operator5'
     *  RelationalOperator: '<S62>/Relational Operator6'
     *  UnitDelay: '<S1>/Unit Delay2'
     */
    if ((Gen2_ref_DWork->x_i && (rtb_Divide2_f > 0.0) &&
         (Gen2_ref_B->BusInput3.traj.rMinCbvAwTvDpCmp >
          Gen2_ref_DWork->UnitDelay2_DSTATE_d)) || (rtb_LogicalOperator && (fabs
          (Gen2_ref_B->Filter4.Switch1) >
          Gen2_ref_B->BusInput3.traj.rMindpdtTvDpCmp)) ||
        Gen2_ref_B->BusInput.tLvrt.bLvrtFlg) {
      delta_y = 0.0;
    } else {
      delta_y = Gen2_ref_B->BusInput3.traj.rGainP2sComp;
    }

    /* End of Switch: '<S62>/Switch2' */
    rtb_Gain_kl = rtb_Sum_c * delta_y;
  }

  /* End of Switch: '<S62>/Switch4' */

  /* BusCreator: '<Root>/Bus Creator' incorporates:
   *  BusCreator: '<S1>/Bus Creator2'
   *  BusCreator: '<S23>/Bus Creator'
   *  DataTypeConversion: '<S1>/Data Type Conversion15'
   *  DataTypeConversion: '<S1>/Data Type Conversion9'
   *  DataTypeConversion: '<S23>/Data Type Conversion5'
   *  DataTypeConversion: '<S78>/Data Type Conversion6'
   *  Outport: '<Root>/dbg'
   * */
  Gen2_ref_Y->dbg.BDC.MP.TVdpFF = (real32_T)rtb_MinMax_a;
  Gen2_ref_Y->dbg.BDC.RL.RLthrsh = (real32_T)rtb_Switch2_jq;
  Gen2_ref_Y->dbg.BDC.FF.CBV_cd = (real32_T)rtb_Sum_mf;
  Gen2_ref_Y->dbg.BDC.FF.TV_cd = (real32_T)rtb_Sum2_a1;

  /* Switch: '<S172>/Switch2' incorporates:
   *  Constant: '<S46>/Constant4'
   *  RelationalOperator: '<S172>/LowerRelop1'
   *  RelationalOperator: '<S172>/UpperRelop'
   *  Switch: '<S172>/Switch'
   */
  if (rtb_DataTypeConversion15 > rtb_Switch13) {
    r = rtb_Switch13;
  } else if (rtb_DataTypeConversion15 < 1.0) {
    /* Switch: '<S172>/Switch' incorporates:
     *  Constant: '<S46>/Constant4'
     */
    r = 1.0;
  } else {
    r = rtb_DataTypeConversion15;
  }

  /* End of Switch: '<S172>/Switch2' */

  /* Saturate: '<S46>/Saturation4' */
  if (Gen2_ref_B->p2s_filt.Switch <= 100000.0) {
    delta_y = 100000.0;
  } else {
    delta_y = Gen2_ref_B->p2s_filt.Switch;
  }

  /* End of Saturate: '<S46>/Saturation4' */

  /* MATLAB Function: '<S46>/engine massflow1' incorporates:
   *  Gain: '<S46>/rpm2rad'
   */
  Gen2_ref_enginemassflow2(delta_y, Gen2_ref_B->T2s_filt.Switch,
    0.10471975511965977 * r, rtb_etaVolConst_lt,
    Gen2_ref_B->BusInput3.eng.rVol_Hub_Eng, &Gen2_ref_B->sf_enginemassflow1_e, inst);

  /* Gain: '<S1>/Gain7' incorporates:
   *  BusCreator: '<S23>/Bus Creator1'
   */
  rtb_Divide2_f = 100000.0 * rtb_Switch2_lu;

  /* MATLAB Function: '<S46>/engine massflow' incorporates:
   *  Gain: '<S46>/rpm2rad1'
   */
  Gen2_ref_enginemassflow(rtb_Divide2_f, Gen2_ref_B->T2s_filt.Switch,
    0.10471975511965977 * rtb_Switch13, rtb_etaVolConst_lt,
    Gen2_ref_B->BusInput3.eng.rVol_Hub_Eng, &Gen2_ref_B->sf_enginemassflow_h, inst);

  /* Gain: '<S46>/rpm2rad2' */
  r = 1.0E-5 * rtb_Divide2_f;

  /* S-Function (sfix_look1_dyn): '<S46>/Lookup Table Dynamic1' */
  /* Dynamic Look-Up Table Block: '<S46>/Lookup Table Dynamic1'
   * Input0  Data Type:  Floating Point real_T
   * Input1  Data Type:  Floating Point real_T
   * Input2  Data Type:  Floating Point real_T
   * Output0 Data Type:  Floating Point real_T
   * Lookup Method: Linear_Endpoint
   *
   */
  LookUp_real_T_real_T( &(rtb_Sum_mf),
                       &Gen2_ref_B->BusInput3.bdcWgv.rRefWGVres_y[0], r,
                       &Gen2_ref_B->BusInput3.bdcWgv.rRefWGVres_x[0], 4U, inst);

  /* Outputs for Atomic SubSystem: '<S46>/cbv tracking1' */
  /* Abs: '<S174>/Abs' */
  rtb_Sum_c = fabs(Gen2_ref_B->BusInput3.bdcWgv.rMaxErrCBVtracking);

  /* Sum: '<S174>/Sum4' incorporates:
   *  Gain: '<S46>/Gain'
   *  Gain: '<S46>/Gain1'
   */
  r = 9.9999999999999991E-6 * rtb_Divide2_f - 9.9999999999999991E-6 *
    Gen2_ref_B->p2s_filt.Switch;

  /* RelationalOperator: '<S174>/Relational Operator2' */
  rtb_LogicalOperator2_ov = (r >
    Gen2_ref_B->BusInput3.bdcWgv.rLimit_p2s_CBVtracking);

  /* Outputs for Atomic SubSystem: '<S174>/TP' */
  /* Product: '<S185>/delta rise limit' incorporates:
   *  SampleTimeMath: '<S185>/sample time'
   *
   * About '<S185>/sample time':
   *  y = K where K = ( w * Ts )
   */
  r = 0.01;

  /* Outputs for Enabled SubSystem: '<S181>/Enabled Subsystem' incorporates:
   *  EnablePort: '<S183>/Enable'
   */
  /* Logic: '<S181>/Logical Operator3' incorporates:
   *  Logic: '<S181>/Logical Operator2'
   *  UnitDelay: '<S181>/Unit Delay2'
   */
  if ((!rtb_LogicalOperator2_ov) && Gen2_ref_DWork->UnitDelay2_DSTATE_b) {
    /* Merge: '<S181>/Merge' incorporates:
     *  Constant: '<S181>/Constant10'
     *  Inport: '<S183>/In1'
     */
    Gen2_ref_B->Merge = 0.0;
  }

  /* End of Logic: '<S181>/Logical Operator3' */
  /* End of Outputs for SubSystem: '<S181>/Enabled Subsystem' */

  /* Outputs for Enabled SubSystem: '<S181>/Enabled Subsystem1' incorporates:
   *  EnablePort: '<S184>/Enable'
   */
  if (rtb_LogicalOperator2_ov) {
    /* Merge: '<S181>/Merge' incorporates:
     *  Inport: '<S184>/In1'
     *  SignalConversion generated from: '<S174>/Bus Selector1'
     */
    Gen2_ref_B->Merge = Gen2_ref_B->BusInput3.bdcWgv.rTi_TP_CBVtracking;
  }

  /* End of Outputs for SubSystem: '<S181>/Enabled Subsystem1' */

  /* UnitDelay: '<S185>/Delay Input2' */
  rtb_Divide2_f = Gen2_ref_DWork->DelayInput2_DSTATE;

  /* Sum: '<S185>/Difference Inputs1' */
  rtb_Sum2_a1 = Gen2_ref_B->Merge - rtb_Divide2_f;

  /* Switch: '<S186>/Switch2' incorporates:
   *  RelationalOperator: '<S186>/LowerRelop1'
   */
  if (!(rtb_Sum2_a1 > 0.01)) {
    /* Switch: '<S186>/Switch' incorporates:
     *  RelationalOperator: '<S186>/UpperRelop'
     */
    if (rtb_Sum2_a1 < -99.990000000000009) {
      r = -99.990000000000009;
    } else {
      r = rtb_Sum2_a1;
    }

    /* End of Switch: '<S186>/Switch' */
  }

  /* End of Switch: '<S186>/Switch2' */

  /* Sum: '<S185>/Difference Inputs2' */
  rtb_Divide2_f += r;

  /* Update for UnitDelay: '<S181>/Unit Delay2' incorporates:
   *  RelationalOperator: '<S181>/Relational Operator3'
   *  SignalConversion generated from: '<S174>/Bus Selector1'
   */
  Gen2_ref_DWork->UnitDelay2_DSTATE_b = (rtb_Divide2_f >=
    Gen2_ref_B->BusInput3.bdcWgv.rTi_TP_CBVtracking);

  /* Update for UnitDelay: '<S185>/Delay Input2' */
  Gen2_ref_DWork->DelayInput2_DSTATE = rtb_Divide2_f;

  /* Logic: '<S174>/Logical Operator5' incorporates:
   *  Constant: '<S179>/Constant'
   *  Constant: '<S182>/Constant'
   *  DataTypeConversion: '<S1>/Data Type Conversion11'
   *  Logic: '<S174>/Logical Operator1'
   *  Logic: '<S174>/Logical Operator4'
   *  Logic: '<S181>/Logical Operator1'
   *  Logic: '<S1>/Logical Operator4'
   *  RelationalOperator: '<S179>/Compare'
   *  RelationalOperator: '<S181>/Relational Operator1'
   *  RelationalOperator: '<S182>/Compare'
   *  SignalConversion generated from: '<S174>/Bus Selector1'
   */
  rtb_LogicalOperator2_ov = ((!Gen2_ref_B->BusInput3.bdcWgv.bTransWGctrl_FF) ||
    (!Gen2_ref_B->BusInput3.bdcWgv.bCBVtracking) ||
    (Gen2_ref_B->BusInput3.eng.rNum_WGV < 0.5) || (!(rtb_Sum1_dh != 0.0)) ||
    ((rtb_Divide2_f > 0.0) && (rtb_Divide2_f <
    Gen2_ref_B->BusInput3.bdcWgv.rTi_TP_CBVtracking)));

  /* End of Outputs for SubSystem: '<S174>/TP' */

  /* DiscreteIntegrator: '<S174>/Discrete-Time Integrator' */
  if (rtb_LogicalOperator2_ov ||
      (Gen2_ref_DWork->DiscreteTimeIntegrator_PrevRe_a != 0)) {
    Gen2_ref_DWork->DiscreteTimeIntegrator_DSTAT_gw = 0.0;
  }

  rtb_DiscreteTimeIntegrator_g3 =
    Gen2_ref_DWork->DiscreteTimeIntegrator_DSTAT_gw;

  /* Sum: '<S174>/Sum' incorporates:
   *  UnitDelay: '<S1>/Unit Delay3'
   */
  rtb_Divide2_f = Gen2_ref_DWork->UnitDelay3_DSTATE_g -
    Gen2_ref_B->BusInput3.bdcWgv.rRefCBVtracking;

  /* Switch: '<S174>/Switch8' incorporates:
   *  Constant: '<S174>/max_PR1'
   */
  if (Gen2_ref_B->TON2.LogicalOperator3) {
    /* Switch: '<S174>/Switch1' incorporates:
     *  Constant: '<S174>/max_PR2'
     *  Constant: '<S174>/max_PR3'
     *  RelationalOperator: '<S174>/Relational Operator1'
     *  Sum: '<S174>/Sum2'
     *  UnitDelay: '<S46>/Unit Delay'
     */
    if (Gen2_ref_DWork->UnitDelay_DSTATE_b >
        Gen2_ref_B->BusInput3.bdcWgv.rPos_max - 0.001) {
      r = 0.0;
    } else {
      r = rtb_Sum_c;
    }

    /* End of Switch: '<S174>/Switch1' */

    /* Switch: '<S180>/Switch2' incorporates:
     *  RelationalOperator: '<S180>/LowerRelop1'
     */
    if (!(rtb_Divide2_f > r)) {
      /* Switch: '<S174>/Switch2' incorporates:
       *  Constant: '<S174>/max_PR2'
       *  Constant: '<S174>/max_PR3'
       *  Gain: '<S174>/Gain'
       *  RelationalOperator: '<S174>/Relational Operator'
       *  Sum: '<S174>/Sum1'
       *  UnitDelay: '<S46>/Unit Delay'
       */
      if (Gen2_ref_DWork->UnitDelay_DSTATE_b <
          Gen2_ref_B->BusInput3.bdcWgv.rPos_min + 0.001) {
        rtb_Sum_c = 0.0;
      } else {
        rtb_Sum_c = -rtb_Sum_c;
      }

      /* End of Switch: '<S174>/Switch2' */

      /* Switch: '<S180>/Switch' incorporates:
       *  RelationalOperator: '<S180>/UpperRelop'
       */
      if (rtb_Divide2_f < rtb_Sum_c) {
        r = rtb_Sum_c;
      } else {
        r = rtb_Divide2_f;
      }

      /* End of Switch: '<S180>/Switch' */
    }

    /* End of Switch: '<S180>/Switch2' */
  } else {
    r = 0.0;
  }

  /* End of Switch: '<S174>/Switch8' */

  /* Product: '<S174>/Divide1' */
  rtb_Divide1_k = rtb_Divide2_f * Gen2_ref_B->BusInput3.bdcWgv.rKpCBVtracking;

  /* Sum: '<S174>/Sum3' incorporates:
   *  DiscreteIntegrator: '<S174>/Discrete-Time Integrator'
   */
  rtb_Sum3_hx = Gen2_ref_DWork->DiscreteTimeIntegrator_DSTAT_gw + rtb_Divide1_k;

  /* Update for DiscreteIntegrator: '<S174>/Discrete-Time Integrator' incorporates:
   *  Product: '<S174>/Divide'
   */
  Gen2_ref_DWork->DiscreteTimeIntegrator_DSTAT_gw +=
    Gen2_ref_B->BusInput3.bdcWgv.rKiCBVtracking * r * 0.01;
  Gen2_ref_DWork->DiscreteTimeIntegrator_PrevRe_a = (int8_T)
    rtb_LogicalOperator2_ov;

  /* End of Outputs for SubSystem: '<S46>/cbv tracking1' */

  /* Sum: '<S46>/Sum4' */
  rtb_Sum_mf += rtb_Sum3_hx;

  /* Product: '<S46>/Divide3' */
  r = Gen2_ref_B->sf_enginemassflow_h.dm_e * rtb_Sum_mf;

  /* Product: '<S46>/Product' incorporates:
   *  Constant: '<S46>/Constant'
   *  Sum: '<S46>/Sum3'
   */
  rtb_Sum_c = (rtb_Sum_mf + 1.0) * Gen2_ref_B->sf_enginemassflow1_e.dm_e;

  /* Gain: '<S1>/Gain8' incorporates:
   *  BusCreator: '<S23>/Bus Creator1'
   */
  rtb_Sum_mf = 100000.0 * Gen2_ref_B->Filter4.Switch1;

  /* DataTypeConversion: '<S175>/Data Type Conversion' */
  rtb_Divide2_f = Gen2_ref_B->BusInput3.bdcWgv.bDynFFwgv_ON;

  /* Sum: '<S175>/Sum3' */
  rtb_Sum2_a1 = rtb_Saturation_cx;

  /* Sum: '<S46>/Sum1' incorporates:
   *  Constant: '<S175>/R_air'
   *  Product: '<S175>/Divide6'
   *  Product: '<S175>/Divide7'
   *  Product: '<S175>/Divide8'
   *  Sum: '<S46>/Sum2'
   */
  rtb_Divide2_f = (rtb_Sum_c - rtb_Sum2_a1 / (287.15 *
    Gen2_ref_B->T2s_filt.Switch) * (rtb_Sum_mf * rtb_Divide2_f)) -
    Gen2_ref_B->sf_enginemassflow_h.dm_e;

  /* Switch: '<S173>/Switch2' incorporates:
   *  RelationalOperator: '<S173>/LowerRelop1'
   */
  if (!(rtb_Divide2_f > r)) {
    /* Switch: '<S173>/Switch' incorporates:
     *  Constant: '<S46>/Constant1'
     *  RelationalOperator: '<S173>/UpperRelop'
     */
    if (rtb_Divide2_f < 0.0) {
      r = 0.0;
    } else {
      r = rtb_Divide2_f;
    }

    /* End of Switch: '<S173>/Switch' */
  }

  /* End of Switch: '<S173>/Switch2' */

  /* Saturate: '<S46>/Saturation5' */
  if (Gen2_ref_B->BusInput3.eng.rNum_WGV > 10.0) {
    rtb_Sum_mf = 10.0;
  } else if (Gen2_ref_B->BusInput3.eng.rNum_WGV < 1.0) {
    rtb_Sum_mf = 1.0;
  } else {
    rtb_Sum_mf = Gen2_ref_B->BusInput3.eng.rNum_WGV;
  }

  /* End of Saturate: '<S46>/Saturation5' */

  /* Product: '<S46>/Divide1' */
  r /= rtb_Sum_mf;

  /* Saturate: '<S46>/Saturation' */
  if (r <= 0.0) {
    rtb_Saturation_cx = 0.0;
  } else {
    rtb_Saturation_cx = r;
  }

  /* End of Saturate: '<S46>/Saturation' */

  /* DataTypeConversion: '<S4>/Data Type Conversion26' */
  r = Gen2_ref_B->BusInput.tPr.rp3HP;

  /* Outputs for Atomic SubSystem: '<S207>/p3LP_filt' */
  /* Gain: '<S4>/bar2Pa7' */
  Gen2_ref_N_TC_HP_filt(100000.0 * r, Gen2_ref_B->BusInput3.inFilt.rTiF_Pr,
                        rtb_bResetBdc, &Gen2_ref_B->p3LP_filt_e,
                        &Gen2_ref_DWork->p3LP_filt_e, inst);

  /* End of Outputs for SubSystem: '<S207>/p3LP_filt' */

  /* Switch: '<S1>/Switch' */
  if (Gen2_ref_B->BusInput3.bdcWgv.bSensorP3 != 0.0) {
    rtb_Divide2_f = Gen2_ref_B->p3LP_filt_e.Switch;
  } else {
    rtb_Divide2_f = Gen2_ref_B->p2s_filt.Switch;
  }

  /* End of Switch: '<S1>/Switch' */

  /* DataTypeConversion: '<S4>/Data Type Conversion7' */
  r = Gen2_ref_B->BusInput.tPr.rp4LP;

  /* Outputs for Atomic SubSystem: '<S208>/p4LP_filt' */
  /* Gain: '<S4>/bar2Pa5' */
  Gen2_ref_N_TC_HP_filt(100000.0 * r, Gen2_ref_B->BusInput3.inFilt.rTiF_Pr,
                        rtb_bResetBdc, &Gen2_ref_B->p4LP_filt,
                        &Gen2_ref_DWork->p4LP_filt, inst);

  /* End of Outputs for SubSystem: '<S208>/p4LP_filt' */

  /* MATLAB Function: '<S46>/MATLAB Function1' incorporates:
   *  Constant: '<S46>/Constant3'
   *  Product: '<S46>/Product1'
   */
  if (rtb_Divide2_f >= Gen2_ref_B->p4LP_filt.Switch) {
    r = Gen2_ref_B->p4LP_filt.Switch / rtb_Divide2_f;
    if ((1.0E-6 >= r) || rtIsNaN(r)) {
      r = 1.0E-6;
    }

    if (1.0 / r <= 1.8929291587378541) {
      u0 = 0.78539816339744828 * Gen2_ref_B->BusInput3.bdcWgv.rDref *
        Gen2_ref_B->BusInput3.bdcWgv.rDref * rtb_Divide2_f / sqrt(287.15 *
        Gen2_ref_B->T2s_filt.Switch) * sqrt((rt_powd_snf(r, 1.4285714285714286, inst)
        - rt_powd_snf(r, 1.7142857142857144, inst)) * 7.0000000000000009);
      if (!(u0 >= 1.0E-6)) {
        u0 = 1.0E-6;
      }

      rtb_Divide2_f = rtb_Saturation_cx / u0;
    } else {
      u0 = 0.78539816339744828 * Gen2_ref_B->BusInput3.bdcWgv.rDref *
        Gen2_ref_B->BusInput3.bdcWgv.rDref * rtb_Divide2_f / sqrt(287.15 *
        Gen2_ref_B->T2s_filt.Switch) * 0.6847314563772704;
      if (!(u0 >= 1.0E-6)) {
        u0 = 1.0E-6;
      }

      rtb_Divide2_f = rtb_Saturation_cx / u0;
    }
  } else {
    rtb_Divide2_f = 0.0;
  }

  /* End of MATLAB Function: '<S46>/MATLAB Function1' */

  /* Saturate: '<S46>/Saturation1' */
  if (rtb_Divide2_f > 1.0) {
    r = 1.0;
  } else if (rtb_Divide2_f < 0.0) {
    r = 0.0;
  } else {
    r = rtb_Divide2_f;
  }

  /* End of Saturate: '<S46>/Saturation1' */
```
